// TIA Portal project "PLC_Project" (V17)

(* hardware
DEVICE "S7-1500/ET200MP station_1"  S7-1500 station
   slot 0: "Rail_0"  Rack  6ES7 590-1***0-0AA0
   slot 1: "PLC_1"  CPU 1512C-1 PN  6ES7 512-1CK01-0AB0  V2.9
      slot 3: "CPU display_1"  6ES7591-1AA00-0AA0
      slot 32768: "PROFINET interface_1"  X1
         slot 32769: "Port_1"  X1 P1
         slot 32770: "Port_2"  X1 P2
      slot 34817: "Virtual CP interface port_1"  Virtual CP interface port  Virtual CP interface port
DEVICE "S7-1200 station_1"  S7-1200 Station
   slot 0: "Rack_0"  S7-1200 Rack  Rack  V1.0
   slot 1: "PLC_2"  CPU 1211C DC/DC/DC  6ES7 211-1AD30-0XB0  V2.2
*)

// ===== PLC "PLC_1"  CPU 1512C-1 PN =====

VAR_GLOBAL   // PLC tag table "ControlStep1"
   "highLevelSilo1" AT %Q0.0 : Bool;
   "lowLevelSilo1" AT %Q0.1 : Bool;
   "highLevelSilo2" AT %Q0.2 : Bool;
   "lowLevelSilo2" AT %Q0.3 : Bool;
   "highLevelSilo3" AT %Q0.4 : Bool;
   "lowLevelSilo3" AT %Q0.5 : Bool;
   "highLevelSilo4" AT %Q0.6 : Bool;
   "lowLevelSilo4" AT %Q0.7 : Bool;
   "highLevelSilo5" AT %Q1.0 : Bool;
   "lowLevelSilo5" AT %Q1.1 : Bool;
   "startPumpSilo1" AT %Q1.2 : Bool;
   "stopPumpSilo1" AT %Q1.3 : Bool;
   "startPumpSilo2" AT %Q1.4 : Bool;
   "stopPumpSilo2" AT %Q1.5 : Bool;
   "startPumpSilo3" AT %Q1.6 : Bool;
   "stopPumpSilo3" AT %Q1.7 : Bool;
   "startPumpSilo4" AT %Q2.0 : Bool;
   "stopPumpSilo4" AT %Q2.1 : Bool;
   "startPumpSilo5" AT %Q2.2 : Bool;
   "stopPumpSilo5" AT %Q2.3 : Bool;
   "errorSilo1" AT %I0.0 : Bool;
   "errorSilo2" AT %I0.1 : Bool;
   "errorSilo3" AT %I0.2 : Bool;
   "errorSilo4" AT %I0.3 : Bool;
   "errorSilo5" AT %I0.4 : Bool;
   "levelSilo1" AT %ID5 : Real;
   "levelSilo2" AT %ID10 : Real;
   "levelSilo3" AT %ID14 : Real;
   "levelSilo4" AT %ID18 : Real;
   "levelSilo5" AT %ID22 : Real;
END_VAR

DATA_BLOCK "Recipe"   // DB1
{ S7_Optimized_Access := 'TRUE' }
VERSION : 0.1
   VAR
      maxLevelSilo1 : Real;   // max cua silo 1
      minLevelSilo1 : Real;   // min cua silo 1
      maxLevelSilo2 : Real;   // max cua silo 2
      minLevelSilo2 : Real;   // min cua silo 2
      maxLevelSilo3 : Real;   // max cua silo 3
      minLevelSilo3 : Real;   // min cua silo 3
      maxLevelSilo4 : Real;   // max cua silo 4
      minLevelSilo4 : Real;   // min cua silo 4
      maxLevelSilo5 : Real;   // max cua silo 5
      minLevelSilo5 : Real;   // min cua silo 5
      weightOfRaw1 : Real;   // khoi luong nguyen lieu 1 can thiet
      weightOfRaw2 : Real;   // khoi luong nguyen lieu 2 can thiet
      weightOfRaw3 : Real;   // khoi luong nguyen lieu 3 can thiet
      weightOfSpice : Real;   // khoi luong gia vi can thiet
      weightOfWater : Real;   // khoi luong nuoc can thiet
      errorWeightRaw1 : Real := 2.5;   // sai so khi do khoi luong nguyen lieu 1
      errorWeightRaw2 : Real := 2.5;   // sai so khi do khoi luong nguyen lieu 2
      errorWeightRaw3 : Real := 2.5;   // sai so khi do khoi luong nguyen lieu 3
      errorWeightSpice : Real := 5.0;   // sai so khi do khoi luong gia vi
      errorWeightWater : Real := 7.0;   // sai so khi do khoi luong nuoc
      openValvePercMin : Real := 10.0;   // % mo van nho nhat de ko gap loi co khi
   END_VAR
BEGIN
END_DATA_BLOCK

DATA_BLOCK "Control_DB"   // DB7
{ S7_Optimized_Access := 'TRUE' }
VERSION : 0.1
// stored: InstanceOfName Control
"Control"
BEGIN
END_DATA_BLOCK

DATA_BLOCK "Process_DB"   // DB8
{ S7_Optimized_Access := 'TRUE' }
VERSION : 0.1
// stored: InstanceOfName Process
"Process"
BEGIN
END_DATA_BLOCK

DATA_BLOCK "BtnControl"   // DB10
{ S7_Optimized_Access := 'TRUE' }
VERSION : 0.1
   VAR
      start : Bool;
      stop : Bool;
      auto : Bool;
      manu : Bool;
      reset : Bool;
      pause : Bool;
      resume : Bool;
      restart : Bool;
      hold : Bool;
      emerg : Bool;
      abort : Bool;
      alarm : Bool;
      error : Bool;
      btn_silo1 : Bool;
      btn_silo2 : Bool;
      btn_silo3 : Bool;
      btn_silo4 : Bool;
      btn_silo5 : Bool;
      btn_Conveyor : Bool;
      btn_scaleRaw1 : Bool;
      btn_scaleRaw2 : Bool;
      btn_scaleRaw3 : Bool;
      btn_scaleSpice : Bool;
      btn_scaleWater : Bool;
      btn_runGrinder : Bool;
      btn_runMixer : Bool;
      btn_dischargeSpice : Bool;
      btn_dischargeWater : Bool;
      btn_dischargeMixer : Bool;
      btn_ResetReady : Bool;
   END_VAR
BEGIN
END_DATA_BLOCK

DATA_BLOCK "Data"   // DB11
{ S7_Optimized_Access := 'TRUE' }
VERSION : 0.1
   VAR
      state : Int;
      "step" : Int;
      mode : Int;
      set : Bool;
      targetBatches : Int;
      currentBatches : Int;
      silo1Ready : Bool;
      silo2Ready : Bool;
      silo3Ready : Bool;
      silo4Ready : Bool;
      silo5Ready : Bool;
      spiceReady : Bool;
      waterReady : Bool;
      rawReady : Bool;
      grindDone : Bool;
      mixDone : Bool;
      productReady : Bool;
      resetReadyState : Bool;
      enaPumpSilo1 : Bool;
      enaPumpSilo2 : Bool;
      enaPumpSilo3 : Bool;
      enaPumpSilo4 : Bool;
      enaPumpSilo5 : Bool;
      enaScaleRaw1 : Bool;
      enaScaleRaw2 : Bool;
      enaScaleRaw3 : Bool;
      enaScaleSpice : Bool;
      enaScaleWater : Bool;
      runConveyor : Bool;
      runGrinder : Bool;
      runMixer : Bool;
      enaDischargeSpice : Bool;
      enaDischargeWater : Bool;
      enaDischargeMixer : Bool;
   END_VAR
BEGIN
END_DATA_BLOCK

// folder: DB

DATA_BLOCK "Phase1_DB"   // DB9
{ S7_Optimized_Access := 'TRUE' }
VERSION : 0.1
// stored: InstanceOfName Phase1
"Phase1"
BEGIN
END_DATA_BLOCK

DATA_BLOCK "Phase2_DB"   // DB12
{ S7_Optimized_Access := 'TRUE' }
VERSION : 0.1
// stored: InstanceOfName Phase2
"Phase2"
BEGIN
END_DATA_BLOCK

DATA_BLOCK "Phase3_DB"   // DB13
{ S7_Optimized_Access := 'TRUE' }
VERSION : 0.1
// stored: InstanceOfName Phase3
"Phase3"
BEGIN
END_DATA_BLOCK

DATA_BLOCK "Phase4_DB"   // DB14
{ S7_Optimized_Access := 'TRUE' }
VERSION : 0.1
// stored: InstanceOfName Phase4
"Phase4"
BEGIN
END_DATA_BLOCK

DATA_BLOCK "Phase5_DB"   // DB15
{ S7_Optimized_Access := 'TRUE' }
VERSION : 0.1
// stored: InstanceOfName Phase5
"Phase5"
BEGIN
END_DATA_BLOCK

DATA_BLOCK "Phase6_DB"   // DB16
{ S7_Optimized_Access := 'TRUE' }
VERSION : 0.1
// stored: InstanceOfName Phase6
"Phase6"
BEGIN
END_DATA_BLOCK

DATA_BLOCK "Phase7_DB"   // DB17
{ S7_Optimized_Access := 'TRUE' }
VERSION : 0.1
// stored: InstanceOfName Phase7
"Phase7"
BEGIN
END_DATA_BLOCK

DATA_BLOCK "Phase8_DB"   // DB18
{ S7_Optimized_Access := 'TRUE' }
VERSION : 0.1
// stored: InstanceOfName Phase8
"Phase8"
BEGIN
END_DATA_BLOCK

DATA_BLOCK "Phase9_DB"   // DB19
{ S7_Optimized_Access := 'TRUE' }
VERSION : 0.1
// stored: InstanceOfName Phase9
"Phase9"
BEGIN
END_DATA_BLOCK

DATA_BLOCK "Phase10_DB"   // DB20
{ S7_Optimized_Access := 'TRUE' }
VERSION : 0.1
// stored: InstanceOfName Phase10
"Phase10"
BEGIN
END_DATA_BLOCK

DATA_BLOCK "Phase11_DB"   // DB21
{ S7_Optimized_Access := 'TRUE' }
VERSION : 0.1
// stored: InstanceOfName Phase11
"Phase11"
BEGIN
END_DATA_BLOCK

DATA_BLOCK "Phase12_DB"   // DB22
{ S7_Optimized_Access := 'TRUE' }
VERSION : 0.1
// stored: InstanceOfName Phase12
"Phase12"
BEGIN
END_DATA_BLOCK

DATA_BLOCK "Phase13_DB"   // DB23
{ S7_Optimized_Access := 'TRUE' }
VERSION : 0.1
// stored: InstanceOfName Phase13
"Phase13"
BEGIN
END_DATA_BLOCK

DATA_BLOCK "Phase14_DB"   // DB24
{ S7_Optimized_Access := 'TRUE' }
VERSION : 0.1
// stored: InstanceOfName Phase14
"Phase14"
BEGIN
END_DATA_BLOCK

DATA_BLOCK "Phase15_DB"   // DB25
{ S7_Optimized_Access := 'TRUE' }
VERSION : 0.1
// stored: InstanceOfName Phase15
"Phase15"
BEGIN
END_DATA_BLOCK

DATA_BLOCK "Phase16_DB"   // DB26
{ S7_Optimized_Access := 'TRUE' }
VERSION : 0.1
// stored: InstanceOfName Phase16
"Phase16"
BEGIN
END_DATA_BLOCK

// folder: System blocks/Program resources

DATA_BLOCK "TON_CheckWeight"   // DB2
{ S7_Optimized_Access := 'TRUE' }
AUTHOR : Simatic
FAMILY : IEC
NAME : IEC_TMR
VERSION : 1.0
// stored: InstanceOfName IEC_TIMER
"IEC_TIMER"
BEGIN
END_DATA_BLOCK

DATA_BLOCK "TON_RunGrinder"   // DB3
{ S7_Optimized_Access := 'TRUE' }
AUTHOR : Simatic
FAMILY : IEC
NAME : IEC_TMR
VERSION : 1.0
// stored: InstanceOfName IEC_TIMER
"IEC_TIMER"
BEGIN
END_DATA_BLOCK

DATA_BLOCK "TON_RunMixer"   // DB4
{ S7_Optimized_Access := 'TRUE' }
AUTHOR : Simatic
FAMILY : IEC
NAME : IEC_TMR
VERSION : 1.0
// stored: InstanceOfName IEC_TIMER
"IEC_TIMER"
BEGIN
END_DATA_BLOCK

DATA_BLOCK "TON_ResetReadyState"   // DB5
{ S7_Optimized_Access := 'TRUE' }
AUTHOR : Simatic
FAMILY : IEC
NAME : IEC_TMR
VERSION : 1.0
// stored: InstanceOfName IEC_TIMER
"IEC_TIMER"
BEGIN
END_DATA_BLOCK

DATA_BLOCK "TP_ResetReadyState"   // DB6
{ S7_Optimized_Access := 'TRUE' }
AUTHOR : Simatic
FAMILY : IEC
NAME : IEC_TMR
VERSION : 1.0
// stored: InstanceOfName IEC_TIMER
"IEC_TIMER"
BEGIN
END_DATA_BLOCK

DATA_BLOCK "TOn_CheckWeightRaw3"   // DB27
{ S7_Optimized_Access := 'TRUE' }
AUTHOR : Simatic
FAMILY : IEC
NAME : IEC_TMR
VERSION : 1.0
// stored: InstanceOfName IEC_TIMER
"IEC_TIMER"
BEGIN
END_DATA_BLOCK

DATA_BLOCK "IEC_Timer_0_DB"   // DB28
{ S7_Optimized_Access := 'TRUE' }
AUTHOR : Simatic
FAMILY : IEC
NAME : IEC_TMR
VERSION : 1.0
// stored: InstanceOfName IEC_TIMER
"IEC_TIMER"
BEGIN
END_DATA_BLOCK

// folder: (top level)

FUNCTION_BLOCK "Control"   // FB1, SCL
{ S7_Optimized_Access := 'TRUE' }
VERSION : 0.1
   VAR_INPUT
      start : Bool;
      stop : Bool;
      auto : Bool;
      manu : Bool;
      reset : Bool;
      pause : Bool;
      resume : Bool;
      restart : Bool;
      hold : Bool;
      emerg : Bool;
      abort : Bool;
      alarm : Bool;
      error : Bool;
   END_VAR
   VAR_IN_OUT
      mode : Int;
      state : Int;
      "step" : Int;
   END_VAR
BEGIN
   //chon che do hoat dong
   IF #state = 0 THEN
       IF (#auto AND #manu) OR (NOT #auto AND NOT #manu) THEN
           #mode := 0;
       ELSE
           IF #auto THEN
               #mode := 1;
           END_IF;
           IF #manu THEN
               #mode := 2;
           END_IF;
       END_IF;
   END_IF;

   IF #mode <> 0 THEN
       CASE #state OF
           0:
               IF #start THEN
                   #state := 1;
               END_IF;
           1:
               IF #abort THEN
                   #state := 2;
               ELSIF #stop THEN
                   #state := 3;
               ELSIF #pause THEN
                   #state := 4;
               ELSIF #hold THEN
                   #state := 5;
               ELSIF #step = 6 THEN
                   #state := 6;
               END_IF;
           2, 3, 6:
               IF #reset THEN
                   #state := 0;
               END_IF;
           4:
               IF #resume THEN
                   #state := 1;
               END_IF;
           5:
               IF #restart THEN
                   #state := 1;
               END_IF;

       END_CASE;
   END_IF;
END_FUNCTION_BLOCK

FUNCTION_BLOCK "Process"   // FB2, SCL
{ S7_Optimized_Access := 'TRUE' }
VERSION : 0.1
   VAR_INPUT
      state : Int;   // trang thai hoat dong
      mode : Int;   // che do hoat dong, 1: auto, 2: manu
      set : Bool;   // tin hieu set cac thong so cai dat
      targetBatches : Int;   // So luong me can lam
      currentBatches : Int;   // So luong me hien tai
      silo1Ready : Bool;   // silo 1 da san sang cung cap nguyen lieu
      silo2Ready : Bool;   // silo 2 da san sang cung cap nguyen lieu
      silo3Ready : Bool;   // silo 3 da san sang cung cap nguyen lieu
      silo4Ready : Bool;   // silo 4 da san sang cung cap gia vi
      silo5Ready : Bool;   // silo 5 da san sang cung cap nuoc
      spiceReady : Bool;   // da can xong gia vi
      waterReady : Bool;   // da can xong nuoc
      rawReady : Bool;   // da can xong va dua nguyen lieu vao bon nghien
      grindDone : Bool;   // da nghien xong nguyen lieu
      mixDone : Bool;   // da tron xong nguyen lieu
      productReady : Bool;
      btn_resetReady : Bool;   // dkhien reset trang thai ready bang tay (mode manu)
      btn_silo1 : Bool;   // dkhien silo bang tay (mode manu)
      btn_silo2 : Bool;   // dkhien silo bang tay (mode manu)
      btn_silo3 : Bool;   // dkhien silo bang tay (mode manu)
      btn_silo4 : Bool;   // dkhien silo bang tay (mode manu)
      btn_silo5 : Bool;   // dkhien silo bang tay (mode manu)
      btn_runConveyor : Bool;   // dkhien can nguyen lieu bang tay (mode manu)
      btn_scaleRaw1 : Bool;   // xa nguyen lieu raw 1 xuong bang tai bang tay (mode manu)
      btn_scaleRaw2 : Bool;   // xa nguyen lieu raw 2 xuong bang tai bang tay (mode manu)
      btn_scaleRaw3 : Bool;   // xa nguyen lieu raw 3 xuong bang tai bang tay (mode manu)
      btn_scaleSpice : Bool;   // dkhien can gia vi bang tay (mode manu)
      btn_scaleWater : Bool;   // dkhien can nuoc bang tay (mode manu)
      btn_runGrinder : Bool;   // dkhien chay may nghien bang tay (mode manu)
      btn_runMixer : Bool;   // dkhien chay may tron bang tay (mode manu)
      btn_DischargeSpice : Bool;   // dkhien van gia vi bang tay (mode manu)
      btn_DischargeWater : Bool;   // dkhien van nuoc bang tay (mode manu)
      btn_DischargeMixer : Bool;   // dkhien van tron bang tay (mode manu)
   END_VAR
   VAR_OUTPUT
      resetReadyState : Bool;   // tiep tuc lam me moi -> reset lai cac bien ready
      enaPumpSilo1 : Bool;   // cho phep bon 1 bat dau hoat dong
      enaPumpSilo2 : Bool;   // cho phep bon 2 bat dau hoat dong
      enaPumpSilo3 : Bool;   // cho phep bon 3 bat dau hoat dong
      enaPumpSilo4 : Bool;   // cho phep bon 4 bat dau hoat dong
      enaPumpSilo5 : Bool;   // cho phep bon 5 bat dau hoat dong
      enaScaleRaw1 : Bool;
      enaScaleRaw2 : Bool;
      enaScaleRaw3 : Bool;
      enaScaleSpice : Bool;   // cho phep can gia vi
      enaScaleWater : Bool;   // cho phep can nuoc
      runConveyor : Bool;   // chay bang tai
      runGrinder : Bool;   // chay may nghien
      runMixer : Bool;   // chay may tron
      enaDischargeSpice : Bool;   // cho phep xa van gia vi vao may tron
      enaDischargeWater : Bool;   // cho phep xa van nuoc vao may tron
      enaDischargeMixer : Bool;   // cho phep xa hon ho[p da tron -> hoan thanh 1 batch
   END_VAR
   VAR_IN_OUT
      "step" : Int;
   END_VAR
BEGIN
   IF #state = 1 AND #mode = 1 AND #set THEN
       IF #step = 0 AND #currentBatches < #targetBatches THEN
           #step := 1;
       END_IF;

       CASE #step OF
           1: 
               #enaPumpSilo1 := TRUE;
               #enaPumpSilo2 := TRUE;
               #enaPumpSilo3 := TRUE;
               #enaPumpSilo4 := TRUE;
               #enaPumpSilo5 := TRUE;
               IF #silo1Ready AND #silo2Ready AND #silo3Ready AND #silo4Ready AND #silo5Ready THEN
                   #enaPumpSilo1 := FALSE;
                   #enaPumpSilo2 := FALSE;
                   #enaPumpSilo3 := FALSE;
                   #enaPumpSilo4 := FALSE;
                   #enaPumpSilo5 := FALSE;
                   #step := 2;
               END_IF;

           2: 
               #runConveyor := TRUE;
               #enaScaleRaw1 := TRUE;
               #enaScaleRaw2 := TRUE;
               #enaScaleRaw3 := TRUE;
               #enaScaleWater := TRUE;
               #enaScaleSpice := TRUE;
               IF #rawReady AND #spiceReady AND #waterReady THEN
                   #runConveyor := FALSE;
                   #enaScaleRaw1 := FALSE;
                   #enaScaleRaw2 := FALSE;
                   #enaScaleRaw3 := FALSE;
                   #enaScaleWater := FALSE;
                   #enaScaleSpice := FALSE;
                   #step := 3;
               END_IF;

           3:
               #runGrinder := TRUE;
               IF #grindDone THEN
                   #runGrinder := FALSE;
                   #step := 4;
               END_IF;

           4: 
               #runMixer := TRUE;
               #enaDischargeWater := TRUE; //cho phep mo van, mo bao nhieu % tuy thuoc vao phase 14, 15 quyet dinh
               #enaDischargeSpice := TRUE;
               IF #mixDone THEN
                   #runMixer := FALSE;
                   #enaDischargeWater := FALSE;
                   #enaDischargeSpice := FALSE;
                   #step := 5;
               END_IF;

           5: 
               #enaDischargeMixer := TRUE;
               IF NOT #productReady THEN
                   #currentBatches := #currentBatches + 1;
                   #enaDischargeMixer := FALSE;
                   #step := 0;
               END_IF;
               // reset cac bien ready ve FALSE trong 1s -> chac chan bien nao cung dc reset
               "TP_ResetReadyState".TP(IN := NOT #productReady,
                                       PT := T#1000ms,
                                       Q => #resetReadyState);
       END_CASE;

   ELSIF #state = 1 AND #mode = 2 AND #set THEN
       #step := 0;
       #resetReadyState := #btn_resetReady;
           //Dk silo
           #enaPumpSilo1 := #btn_silo1;
           #enaPumpSilo2 := #btn_silo2;
           #enaPumpSilo3 := #btn_silo3;
           #enaPumpSilo4 := #btn_silo4;
           #enaPumpSilo5 := #btn_silo5;

           //Dk can va bang tai 
           #runConveyor := #btn_runConveyor;
           #enaScaleRaw1 := #btn_scaleRaw1;
           #enaScaleRaw2 := #btn_scaleRaw2;
           #enaScaleRaw3 := #btn_scaleRaw3;
           #enaScaleWater := #btn_scaleWater;
           #enaScaleSpice := #btn_scaleWater;

           //Dk may nghien va may tron
           #runGrinder := #btn_runGrinder;
           #runMixer := #btn_runMixer;

           //Dong/mo van
           #enaDischargeWater := #btn_DischargeWater;
           #enaDischargeSpice := #btn_DischargeSpice;
           #enaDischargeMixer := #btn_DischargeMixer;
   END_IF;
END_FUNCTION_BLOCK

ORGANIZATION_BLOCK "Main"   // OB1, LAD, ProgramCycle
TITLE = "Main Program Sweep (Cycle)"
{ S7_Optimized_Access := 'TRUE' }
VERSION : 0.1
   VAR_INPUT
      Initial_Call : Bool;   // Initial call of this OB
      Remanence : Bool;   // =True, if remanent data are available
   END_VAR
   VAR_TEMP   // added for the SCL form of the ladder/FBD networks
      _w1 : Bool;
      _w2 : Bool;
   END_VAR
BEGIN

REGION Network 1
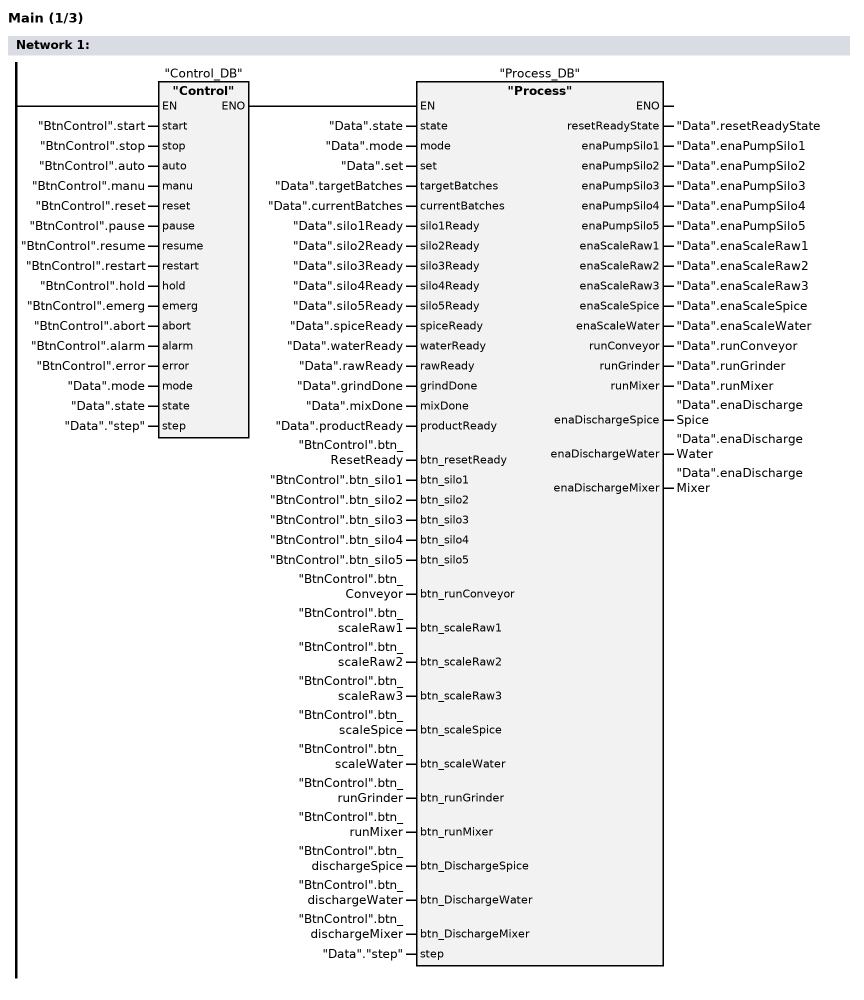
   RUNG wire#powerrail
      "Control_DB"(start := "BtnControl".start, stop := "BtnControl".stop, auto := "BtnControl".auto, manu := "BtnControl".manu, reset := "BtnControl".reset, pause := "BtnControl".pause, resume := "BtnControl".resume, restart := "BtnControl".restart, hold := "BtnControl".hold, emerg := "BtnControl".emerg, abort := "BtnControl".abort, alarm := "BtnControl".alarm, error := "BtnControl".error, mode := "Data".mode, state := "Data".state, "step" := "Data"."step")
      "Process_DB"(state := "Data".state, mode := "Data".mode, set := "Data".set, targetBatches := "Data".targetBatches, currentBatches := "Data".currentBatches, silo1Ready := "Data".silo1Ready, silo2Ready := "Data".silo2Ready, silo3Ready := "Data".silo3Ready, silo4Ready := "Data".silo4Ready, silo5Ready := "Data".silo5Ready, spiceReady := "Data".spiceReady, waterReady := "Data".waterReady, rawReady := "Data".rawReady, grindDone := "Data".grindDone, mixDone := "Data".mixDone, productReady := "Data".productReady, btn_resetReady := "BtnControl".btn_ResetReady, btn_silo1 := "BtnControl".btn_silo1, btn_silo2 := "BtnControl".btn_silo2, btn_silo3 := "BtnControl".btn_silo3, btn_silo4 := "BtnControl".btn_silo4, btn_silo5 := "BtnControl".btn_silo5, btn_runConveyor := "BtnControl".btn_Conveyor, btn_scaleRaw1 := "BtnControl".btn_scaleRaw1, btn_scaleRaw2 := "BtnControl".btn_scaleRaw2, btn_scaleRaw3 := "BtnControl".btn_scaleRaw3, btn_scaleSpice := "BtnControl".btn_scaleSpice, btn_scaleWater := "BtnControl".btn_scaleWater, btn_runGrinder := "BtnControl".btn_runGrinder, btn_runMixer := "BtnControl".btn_runMixer, btn_DischargeSpice := "BtnControl".btn_dischargeSpice, btn_DischargeWater := "BtnControl".btn_dischargeWater, btn_DischargeMixer := "BtnControl".btn_dischargeMixer, "step" := "Data"."step", resetReadyState => "Data".resetReadyState, enaPumpSilo1 => "Data".enaPumpSilo1, enaPumpSilo2 => "Data".enaPumpSilo2, enaPumpSilo3 => "Data".enaPumpSilo3, enaPumpSilo4 => "Data".enaPumpSilo4, enaPumpSilo5 => "Data".enaPumpSilo5, enaScaleRaw1 => "Data".enaScaleRaw1, enaScaleRaw2 => "Data".enaScaleRaw2, enaScaleRaw3 => "Data".enaScaleRaw3, enaScaleSpice => "Data".enaScaleSpice, enaScaleWater => "Data".enaScaleWater, runConveyor => "Data".runConveyor, runGrinder => "Data".runGrinder, runMixer => "Data".runMixer, enaDischargeSpice => "Data".enaDischargeSpice, enaDischargeWater => "Data".enaDischargeWater, enaDischargeMixer => "Data".enaDischargeMixer)
   END_RUNG
   // the same network as SCL:
   "Control_DB"(start := "BtnControl".start,   // "Control"
                stop := "BtnControl".stop,
                auto := "BtnControl".auto,
                manu := "BtnControl".manu,
                reset := "BtnControl".reset,
                pause := "BtnControl".pause,
                resume := "BtnControl".resume,
                restart := "BtnControl".restart,
                hold := "BtnControl".hold,
                emerg := "BtnControl".emerg,
                abort := "BtnControl".abort,
                alarm := "BtnControl".alarm,
                error := "BtnControl".error,
                mode := "Data".mode,
                state := "Data".state,
                "step" := "Data"."step",
                ENO => #_w1);
   IF #_w1 THEN
       "Process_DB"(state := "Data".state,   // "Process"
                    mode := "Data".mode,
                    set := "Data".set,
                    targetBatches := "Data".targetBatches,
                    currentBatches := "Data".currentBatches,
                    silo1Ready := "Data".silo1Ready,
                    silo2Ready := "Data".silo2Ready,
                    silo3Ready := "Data".silo3Ready,
                    silo4Ready := "Data".silo4Ready,
                    silo5Ready := "Data".silo5Ready,
                    spiceReady := "Data".spiceReady,
                    waterReady := "Data".waterReady,
                    rawReady := "Data".rawReady,
                    grindDone := "Data".grindDone,
                    mixDone := "Data".mixDone,
                    productReady := "Data".productReady,
                    btn_resetReady := "BtnControl".btn_ResetReady,
                    btn_silo1 := "BtnControl".btn_silo1,
                    btn_silo2 := "BtnControl".btn_silo2,
                    btn_silo3 := "BtnControl".btn_silo3,
                    btn_silo4 := "BtnControl".btn_silo4,
                    btn_silo5 := "BtnControl".btn_silo5,
                    btn_runConveyor := "BtnControl".btn_Conveyor,
                    btn_scaleRaw1 := "BtnControl".btn_scaleRaw1,
                    btn_scaleRaw2 := "BtnControl".btn_scaleRaw2,
                    btn_scaleRaw3 := "BtnControl".btn_scaleRaw3,
                    btn_scaleSpice := "BtnControl".btn_scaleSpice,
                    btn_scaleWater := "BtnControl".btn_scaleWater,
                    btn_runGrinder := "BtnControl".btn_runGrinder,
                    btn_runMixer := "BtnControl".btn_runMixer,
                    btn_DischargeSpice := "BtnControl".btn_dischargeSpice,
                    btn_DischargeWater := "BtnControl".btn_dischargeWater,
                    btn_DischargeMixer := "BtnControl".btn_dischargeMixer,
                    "step" := "Data"."step",
                    resetReadyState => "Data".resetReadyState,
                    enaPumpSilo1 => "Data".enaPumpSilo1,
                    enaPumpSilo2 => "Data".enaPumpSilo2,
                    enaPumpSilo3 => "Data".enaPumpSilo3,
                    enaPumpSilo4 => "Data".enaPumpSilo4,
                    enaPumpSilo5 => "Data".enaPumpSilo5,
                    enaScaleRaw1 => "Data".enaScaleRaw1,
                    enaScaleRaw2 => "Data".enaScaleRaw2,
                    enaScaleRaw3 => "Data".enaScaleRaw3,
                    enaScaleSpice => "Data".enaScaleSpice,
                    enaScaleWater => "Data".enaScaleWater,
                    runConveyor => "Data".runConveyor,
                    runGrinder => "Data".runGrinder,
                    runMixer => "Data".runMixer,
                    enaDischargeSpice => "Data".enaDischargeSpice,
                    enaDischargeWater => "Data".enaDischargeWater,
                    enaDischargeMixer => "Data".enaDischargeMixer);
   END_IF;
END_REGION

REGION Network 2
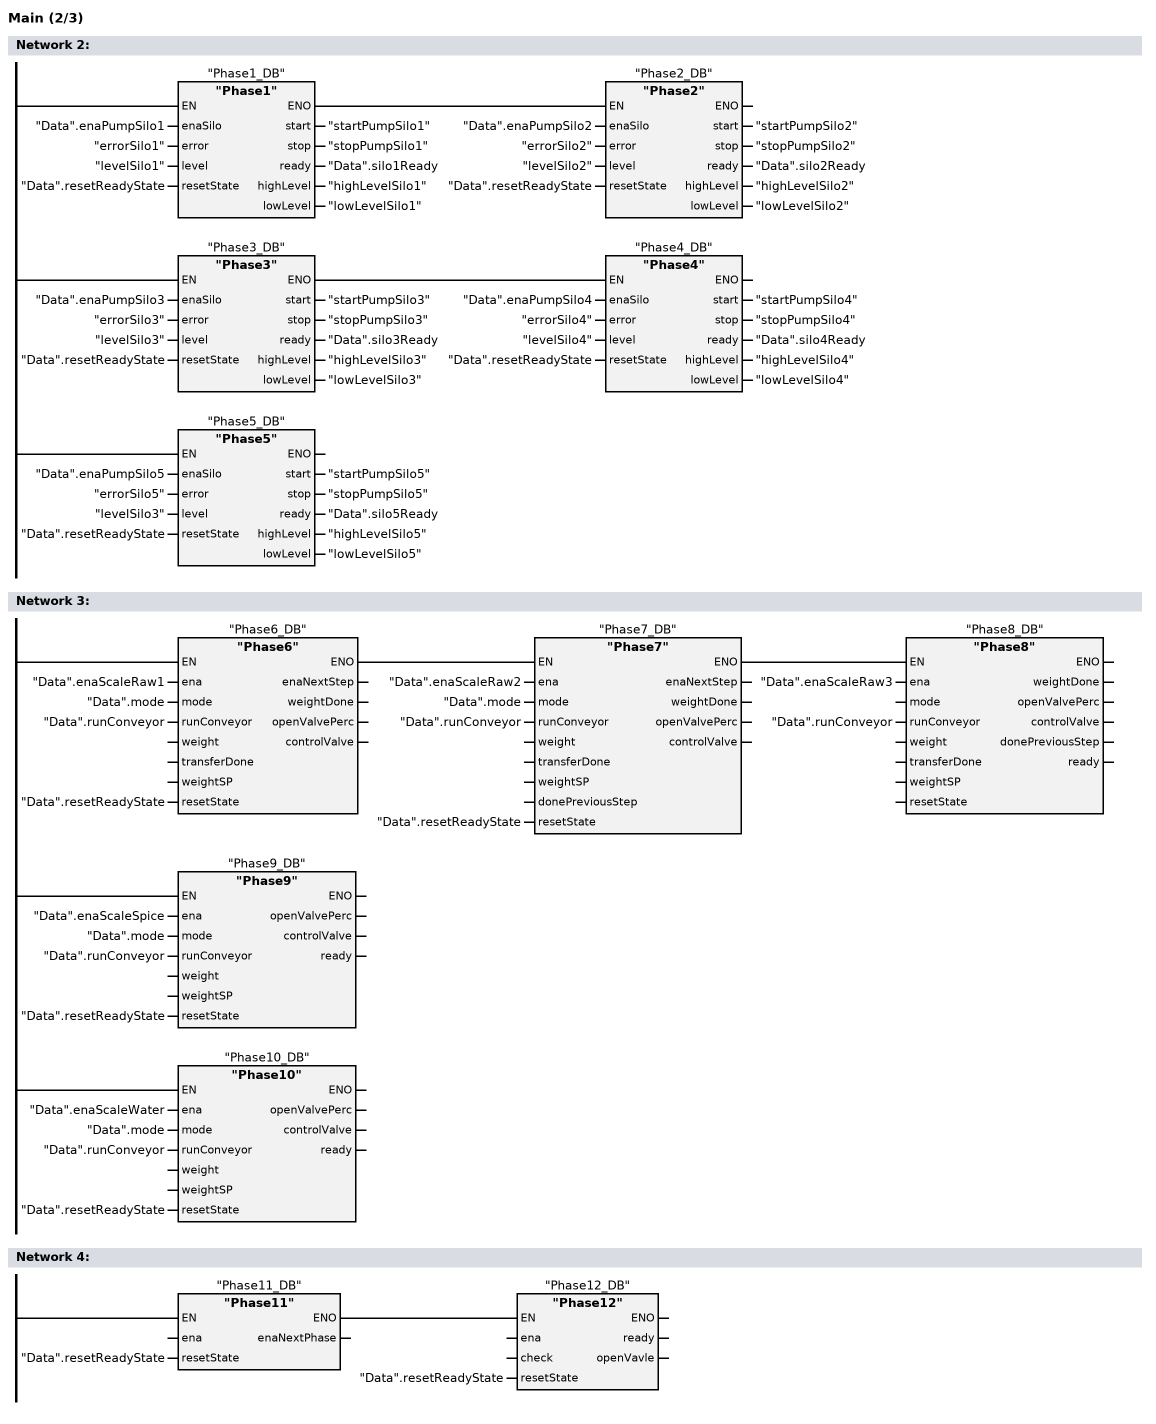
   RUNG wire#powerrail
      "Phase1_DB"(enaSilo := "Data".enaPumpSilo1, error := "errorSilo1", level := "levelSilo1", resetState := "Data".resetReadyState, start => "startPumpSilo1", stop => "stopPumpSilo1", ready => "Data".silo1Ready, highLevel => "highLevelSilo1", lowLevel => "lowLevelSilo1")
      "Phase2_DB"(enaSilo := "Data".enaPumpSilo2, error := "errorSilo2", level := "levelSilo2", resetState := "Data".resetReadyState, start => "startPumpSilo2", stop => "stopPumpSilo2", ready => "Data".silo2Ready, highLevel => "highLevelSilo2", lowLevel => "lowLevelSilo2")
   END_RUNG
   RUNG wire#powerrail
      "Phase3_DB"(enaSilo := "Data".enaPumpSilo3, error := "errorSilo3", level := "levelSilo3", resetState := "Data".resetReadyState, start => "startPumpSilo3", stop => "stopPumpSilo3", ready => "Data".silo3Ready, highLevel => "highLevelSilo3", lowLevel => "lowLevelSilo3")
      "Phase4_DB"(enaSilo := "Data".enaPumpSilo4, error := "errorSilo4", level := "levelSilo4", resetState := "Data".resetReadyState, start => "startPumpSilo4", stop => "stopPumpSilo4", ready => "Data".silo4Ready, highLevel => "highLevelSilo4", lowLevel => "lowLevelSilo4")
   END_RUNG
   RUNG wire#powerrail
      "Phase5_DB"(enaSilo := "Data".enaPumpSilo5, error := "errorSilo5", level := "levelSilo3", resetState := "Data".resetReadyState, start => "startPumpSilo5", stop => "stopPumpSilo5", ready => "Data".silo5Ready, highLevel => "highLevelSilo5", lowLevel => "lowLevelSilo5")
   END_RUNG
   // the same network as SCL:
   "Phase1_DB"(enaSilo := "Data".enaPumpSilo1,   // "Phase1"
               error := "errorSilo1",
               level := "levelSilo1",
               resetState := "Data".resetReadyState,
               start => "startPumpSilo1",
               stop => "stopPumpSilo1",
               ready => "Data".silo1Ready,
               highLevel => "highLevelSilo1",
               lowLevel => "lowLevelSilo1",
               ENO => #_w1);
   IF #_w1 THEN
       "Phase2_DB"(enaSilo := "Data".enaPumpSilo2,   // "Phase2"
                   error := "errorSilo2",
                   level := "levelSilo2",
                   resetState := "Data".resetReadyState,
                   start => "startPumpSilo2",
                   stop => "stopPumpSilo2",
                   ready => "Data".silo2Ready,
                   highLevel => "highLevelSilo2",
                   lowLevel => "lowLevelSilo2");
   END_IF;
   "Phase3_DB"(enaSilo := "Data".enaPumpSilo3,   // "Phase3"
               error := "errorSilo3",
               level := "levelSilo3",
               resetState := "Data".resetReadyState,
               start => "startPumpSilo3",
               stop => "stopPumpSilo3",
               ready => "Data".silo3Ready,
               highLevel => "highLevelSilo3",
               lowLevel => "lowLevelSilo3",
               ENO => #_w2);
   IF #_w2 THEN
       "Phase4_DB"(enaSilo := "Data".enaPumpSilo4,   // "Phase4"
                   error := "errorSilo4",
                   level := "levelSilo4",
                   resetState := "Data".resetReadyState,
                   start => "startPumpSilo4",
                   stop => "stopPumpSilo4",
                   ready => "Data".silo4Ready,
                   highLevel => "highLevelSilo4",
                   lowLevel => "lowLevelSilo4");
   END_IF;
   "Phase5_DB"(enaSilo := "Data".enaPumpSilo5,   // "Phase5"
               error := "errorSilo5",
               level := "levelSilo3",
               resetState := "Data".resetReadyState,
               start => "startPumpSilo5",
               stop => "stopPumpSilo5",
               ready => "Data".silo5Ready,
               highLevel => "highLevelSilo5",
               lowLevel => "lowLevelSilo5");
END_REGION

REGION Network 3
   RUNG wire#powerrail
      "Phase6_DB"(ena := "Data".enaScaleRaw1, mode := "Data".mode, runConveyor := "Data".runConveyor, weight :=, transferDone :=, weightSP :=, resetState := "Data".resetReadyState, enaNextStep =>, weightDone =>, openValvePerc =>, controlValve =>)
      "Phase7_DB"(ena := "Data".enaScaleRaw2, mode := "Data".mode, runConveyor := "Data".runConveyor, weight :=, transferDone :=, weightSP :=, donePreviousStep :=, resetState := "Data".resetReadyState, enaNextStep =>, weightDone =>, openValvePerc =>, controlValve =>)
      "Phase8_DB"(ena := "Data".enaScaleRaw3, mode :=, runConveyor := "Data".runConveyor, weight :=, transferDone :=, weightSP :=, resetState :=, weightDone =>, openValvePerc =>, controlValve =>, donePreviousStep =>, ready =>)
   END_RUNG
   RUNG wire#powerrail
      "Phase9_DB"(ena := "Data".enaScaleSpice, mode := "Data".mode, runConveyor := "Data".runConveyor, weight :=, weightSP :=, resetState := "Data".resetReadyState, openValvePerc =>, controlValve =>, ready =>)
   END_RUNG
   RUNG wire#powerrail
      "Phase10_DB"(ena := "Data".enaScaleWater, mode := "Data".mode, runConveyor := "Data".runConveyor, weight :=, weightSP :=, resetState := "Data".resetReadyState, openValvePerc =>, controlValve =>, ready =>)
   END_RUNG
   // the same network as SCL:
   "Phase6_DB"(ena := "Data".enaScaleRaw1,   // "Phase6"
               mode := "Data".mode,
               runConveyor := "Data".runConveyor,
               resetState := "Data".resetReadyState,
               ENO => #_w1);
   "Phase7_DB"(EN := #_w1,   // "Phase7"
               ena := "Data".enaScaleRaw2,
               mode := "Data".mode,
               runConveyor := "Data".runConveyor,
               resetState := "Data".resetReadyState,
               ENO => #_w2);
   IF #_w2 THEN
       "Phase8_DB"(ena := "Data".enaScaleRaw3, runConveyor := "Data".runConveyor);   // "Phase8"
   END_IF;
   "Phase9_DB"(ena := "Data".enaScaleSpice,   // "Phase9"
               mode := "Data".mode,
               runConveyor := "Data".runConveyor,
               resetState := "Data".resetReadyState);
   "Phase10_DB"(ena := "Data".enaScaleWater,   // "Phase10"
                mode := "Data".mode,
                runConveyor := "Data".runConveyor,
                resetState := "Data".resetReadyState);
END_REGION

REGION Network 4
   RUNG wire#powerrail
      "Phase11_DB"(ena :=, resetState := "Data".resetReadyState, enaNextPhase =>)
      "Phase12_DB"(ena :=, check :=, resetState := "Data".resetReadyState, ready =>, openVavle =>)
   END_RUNG
   // the same network as SCL:
   "Phase11_DB"(resetState := "Data".resetReadyState, ENO => #_w1);   // "Phase11"
   IF #_w1 THEN
       "Phase12_DB"(resetState := "Data".resetReadyState);   // "Phase12"
   END_IF;
END_REGION

REGION Network 5
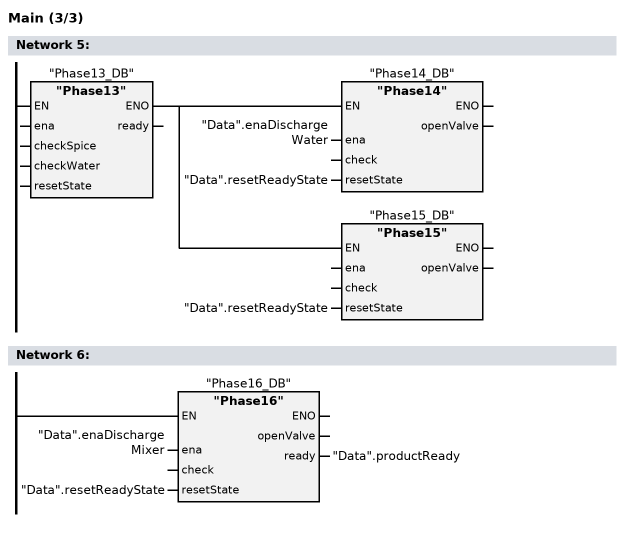
   RUNG wire#powerrail
      "Phase13_DB"(ena :=, checkSpice :=, checkWater :=, resetState :=, ready =>)
      wire#w1
      "Phase14_DB"(ena := "Data".enaDischargeWater, check :=, resetState := "Data".resetReadyState, openValve =>)
   END_RUNG
   RUNG wire#w1
      "Phase15_DB"(ena :=, check :=, resetState := "Data".resetReadyState, openValve =>)
   END_RUNG
   // the same network as SCL:
   "Phase13_DB"(ENO => #_w1);   // "Phase13"
   IF #_w1 THEN
       "Phase14_DB"(ena := "Data".enaDischargeWater, resetState := "Data".resetReadyState);   // "Phase14"
       "Phase15_DB"(resetState := "Data".resetReadyState);   // "Phase15"
   END_IF;
END_REGION

REGION Network 6
   RUNG wire#powerrail
      "Phase16_DB"(ena := "Data".enaDischargeMixer, check :=, resetState := "Data".resetReadyState, openValve =>, ready => "Data".productReady)
   END_RUNG
   // the same network as SCL:
   "Phase16_DB"(ena := "Data".enaDischargeMixer,   // "Phase16"
                resetState := "Data".resetReadyState,
                ready => "Data".productReady);
END_REGION
END_ORGANIZATION_BLOCK

// folder: Unit1(prepareSilo1_Raw)

FUNCTION_BLOCK "Phase1"   // FB3, SCL
{ S7_Optimized_Access := 'TRUE' }
VERSION : 0.1
   VAR_INPUT
      enaSilo : Bool;
      error : Bool;
      level : Real;
      resetState : Bool;
   END_VAR
   VAR_OUTPUT
      start : Bool;
      stop : Bool;
      ready : Bool;
      highLevel : Bool;
      lowLevel : Bool;
   END_VAR
BEGIN
   #highLevel := #level >= "Recipe".maxLevelSilo1;
   #lowLevel := #level <= "Recipe".minLevelSilo1;
   #start := #enaSilo AND #lowLevel;
   #stop := #highLevel OR #error;
   #ready := NOT #highLevel AND NOT #lowLevel;
   IF #resetState THEN
       #ready := FALSE;
   END_IF;
END_FUNCTION_BLOCK

// folder: Unit10(mixAndDone)

FUNCTION_BLOCK "Phase13"   // FB15, SCL
{ S7_Optimized_Access := 'TRUE' }
VERSION : 0.1
   VAR_INPUT
      ena : Bool;   // cho phep hoat dong mixer
      checkSpice : Bool;   // ktra da co du gia vi trong bon chua
      checkWater : Bool;   // ktra da co du nuoc trong bon chua
      resetState : Bool;
   END_VAR
   VAR_OUTPUT
      ready : Bool;
   END_VAR
   VAR CONSTANT
      "time" : Time := T#10s;
   END_VAR
BEGIN
       "TON_RunMixer".TON(IN := #ena AND #checkSpice AND #checkWater,
                          PT := #time,
                          Q => #ready);
       IF #resetState THEN
           #ready := FALSE;
       END_IF;
END_FUNCTION_BLOCK

FUNCTION_BLOCK "Phase14"   // FB16, SCL
{ S7_Optimized_Access := 'TRUE' }
VERSION : 0.1
   VAR_INPUT
      ena : Bool;
      check : Bool;   // ktra bon con gia vi ko
      resetState : Bool;
   END_VAR
   VAR_OUTPUT
      openValve : Bool;
   END_VAR
BEGIN
   IF #ena THEN
       #openValve := TRUE;
       IF NOT #check THEN
           #openValve := FALSE;
       END_IF;
   END_IF;
END_FUNCTION_BLOCK

FUNCTION_BLOCK "Phase15"   // FB17, SCL
{ S7_Optimized_Access := 'TRUE' }
VERSION : 0.1
   VAR_INPUT
      ena : Bool;
      check : Bool;   // ktra bon con nuoc ko
      resetState : Bool;
   END_VAR
   VAR_OUTPUT
      openValve : Bool;
   END_VAR
BEGIN
   IF #ena THEN
       #openValve := TRUE;
       IF NOT #check THEN
           #openValve := FALSE;
       END_IF;
   END_IF;
END_FUNCTION_BLOCK

FUNCTION_BLOCK "Phase16"   // FB18, SCL
{ S7_Optimized_Access := 'TRUE' }
VERSION : 0.1
   VAR_INPUT
      ena : Bool;
      check : Bool;   // ktra hon hop con trong bon ko
      resetState : Bool;
   END_VAR
   VAR_OUTPUT
      openValve : Bool;
      ready : Bool;
   END_VAR
BEGIN
   IF #ena THEN
       #openValve := TRUE;
       IF NOT #check THEN
           #openValve := FALSE;
           #ready := TRUE;
       END_IF;
   END_IF;

   IF #resetState THEN
       #ready := FALSE;
   END_IF;
END_FUNCTION_BLOCK

// folder: Unit2(prepareSilo2_Raw)

FUNCTION_BLOCK "Phase2"   // FB4, SCL
{ S7_Optimized_Access := 'TRUE' }
VERSION : 0.1
   VAR_INPUT
      enaSilo : Bool;
      error : Bool;
      level : Real;
      resetState : Bool;
   END_VAR
   VAR_OUTPUT
      start : Bool;
      stop : Bool;
      ready : Bool;
      highLevel : Bool;
      lowLevel : Bool;
   END_VAR
BEGIN
   #highLevel := #level >= "Recipe".maxLevelSilo2;
   #lowLevel := #level <= "Recipe".minLevelSilo2;
   #start := #enaSilo AND #lowLevel;
   #stop := #highLevel OR #error;
   #ready := NOT #highLevel AND NOT #lowLevel;
   IF #resetState THEN
       #ready := FALSE;
   END_IF;
END_FUNCTION_BLOCK

// folder: Unit3(prepareSilo3_Raw)

FUNCTION_BLOCK "Phase3"   // FB5, SCL
{ S7_Optimized_Access := 'TRUE' }
VERSION : 0.1
   VAR_INPUT
      enaSilo : Bool;
      error : Bool;
      level : Real;
      resetState : Bool;
   END_VAR
   VAR_OUTPUT
      start : Bool;
      stop : Bool;
      ready : Bool;
      highLevel : Bool;
      lowLevel : Bool;
   END_VAR
BEGIN
   #highLevel := #level >= "Recipe".maxLevelSilo3;
   #lowLevel := #level <= "Recipe".minLevelSilo3;
   #start := #enaSilo AND #lowLevel;
   #stop := #highLevel OR #error;
   #ready := NOT #highLevel AND NOT #lowLevel;
   IF #resetState THEN
       #ready := FALSE;
   END_IF;
END_FUNCTION_BLOCK

// folder: Unit4(prepareSilo4_Spice)

FUNCTION_BLOCK "Phase4"   // FB6, SCL
{ S7_Optimized_Access := 'TRUE' }
VERSION : 0.1
   VAR_INPUT
      enaSilo : Bool;
      error : Bool;
      level : Real;
      resetState : Bool;
   END_VAR
   VAR_OUTPUT
      start : Bool;
      stop : Bool;
      ready : Bool;
      highLevel : Bool;
      lowLevel : Bool;
   END_VAR
BEGIN
   #highLevel := #level >= "Recipe".maxLevelSilo4;
   #lowLevel := #level <= "Recipe".minLevelSilo4;
   #start := #enaSilo AND #lowLevel;
   #stop := #highLevel OR #error;
   #ready := NOT #highLevel AND NOT #lowLevel;
   IF #resetState THEN
       #ready := FALSE;
   END_IF;
END_FUNCTION_BLOCK

// folder: Unit5(prepareSilo5_Water)

FUNCTION_BLOCK "Phase5"   // FB7, SCL
{ S7_Optimized_Access := 'TRUE' }
VERSION : 0.1
   VAR_INPUT
      enaSilo : Bool;
      error : Bool;
      level : Real;
      resetState : Bool;
   END_VAR
   VAR_OUTPUT
      start : Bool;
      stop : Bool;
      ready : Bool;
      highLevel : Bool;
      lowLevel : Bool;
   END_VAR
BEGIN
   #highLevel := #level >= "Recipe".maxLevelSilo5;
   #lowLevel := #level <= "Recipe".minLevelSilo5;
   #start := #enaSilo AND #lowLevel;
   #stop := #highLevel OR #error;
   #ready := NOT #highLevel AND NOT #lowLevel;
   IF #resetState THEN
       #ready := FALSE;
   END_IF;
END_FUNCTION_BLOCK

// folder: Unit6(scaleAndTransferRaw)

FUNCTION_BLOCK "Phase6"   // FB8, SCL
{ S7_Optimized_Access := 'TRUE' }
VERSION : 0.1
   VAR_INPUT
      ena : Bool;
      mode : Int;
      runConveyor : Bool;
      weight : Real;
      transferDone : Bool;
      weightSP : Real;
      resetState : Bool;
   END_VAR
   VAR_OUTPUT
      enaNextStep : Bool;
      weightDone : Bool;
      openValvePerc : Real;
      controlValve : Real;
   END_VAR
   VAR CONSTANT
      factor : Real := 10.0;
      "time" : Time := T#300ms;
   END_VAR
BEGIN
   IF #ena AND NOT #weightDone AND #mode = 1 THEN
       IF ABS_REAL(#weight - #weightSP) > "Recipe".errorWeightRaw1 * #factor THEN
           #openValvePerc := 100;
       ELSE
           #openValvePerc := ABS_REAL(#weight - #weightSP)/"Recipe".errorWeightRaw1 * #factor;
           IF #openValvePerc < "Recipe".openValvePercMin THEN
               #openValvePerc := "Recipe".openValvePercMin;
           END_IF;
       END_IF;
   ELSIF #ena AND #mode = 2 THEN
       #openValvePerc := 50;
   ELSE
       #openValvePerc := 0;
   END_IF;

   IF ABS_REAL( #weight - #weightSP) <= "Recipe".errorWeightRaw1 THEN
       #weightDone := TRUE;
   END_IF;

   IF #weightDone  AND #transferDone THEN
       #enaNextStep := TRUE;
   END_IF;
   IF #resetState THEN
       #enaNextStep := FALSE;
   END_IF;
END_FUNCTION_BLOCK

FUNCTION_BLOCK "Phase7"   // FB9, SCL
{ S7_Optimized_Access := 'TRUE' }
VERSION : 0.1
   VAR_INPUT
      ena : Bool;
      mode : Int;
      runConveyor : Bool;
      weight : Real;
      transferDone : Bool;
      weightSP : Real;
      donePreviousStep : Bool;
      resetState : Bool;
   END_VAR
   VAR_OUTPUT
      enaNextStep : Bool;
      weightDone : Bool;
      openValvePerc : Real;
      controlValve : Real;
   END_VAR
   VAR CONSTANT
      factor : Real := 10.0;
      "time" : Time := T#300ms;
   END_VAR
BEGIN
   IF #ena AND NOT #weightDone AND #mode = 1 AND #donePreviousStep THEN
       IF ABS_REAL(#weight - #weightSP) > "Recipe".errorWeightRaw2 * #factor THEN
           #openValvePerc := 100;
       ELSE
           #openValvePerc := ABS_REAL(#weight - #weightSP) / "Recipe".errorWeightRaw2 * #factor;
           IF #openValvePerc < "Recipe".openValvePercMin THEN
               #openValvePerc := "Recipe".openValvePercMin;
           END_IF;
       END_IF;
   ELSIF #ena AND #mode = 2 THEN
       #openValvePerc := 50;
   ELSE
       #openValvePerc := 0;
   END_IF;

   IF ABS_REAL(#weight - #weightSP) <= "Recipe".errorWeightRaw1 THEN
       #weightDone := TRUE;
   END_IF;

   IF #weightDone AND #transferDone THEN
       #enaNextStep := TRUE;
   END_IF;
   IF #resetState THEN
       #enaNextStep := FALSE;
   END_IF;
END_FUNCTION_BLOCK

FUNCTION_BLOCK "Phase8"   // FB10, SCL
{ S7_Optimized_Access := 'TRUE' }
VERSION : 0.1
   VAR_INPUT
      ena : Bool;
      mode : Int;
      runConveyor : Bool;
      weight : Real;
      transferDone : Bool;
      weightSP : Real;
      resetState : Bool;
   END_VAR
   VAR_OUTPUT
      weightDone : Bool;
      openValvePerc : Real;
      controlValve : Real;
      donePreviousStep : Bool;
      ready : Bool;
   END_VAR
   VAR CONSTANT
      factor : Real := 10.0;
      "time" : Time := T#300ms;
   END_VAR
BEGIN
   IF #ena AND NOT #weightDone AND #mode = 1 AND #donePreviousStep THEN
       IF ABS_REAL(#weight - #weightSP) > "Recipe".errorWeightRaw3 * #factor THEN
           #openValvePerc := 100;
       ELSE
           #openValvePerc := ABS_REAL(#weight - #weightSP) / "Recipe".errorWeightRaw3 * #factor;
           IF #openValvePerc < "Recipe".openValvePercMin THEN
               #openValvePerc := "Recipe".openValvePercMin;
           END_IF;
       END_IF;
   ELSIF #ena AND #mode = 2 THEN
       #openValvePerc := 50;
   ELSE
       #openValvePerc := 0;
   END_IF;

   IF ABS_REAL(#weight - #weightSP) <= "Recipe".errorWeightRaw1 THEN
       #weightDone := TRUE;
   END_IF;

   IF #weightDone AND #transferDone THEN
       #ready := TRUE;
   END_IF;
   IF #resetState THEN
       #ready := FALSE;
   END_IF;
END_FUNCTION_BLOCK

// folder: Unit7(scaleSpice)

FUNCTION_BLOCK "Phase9"   // FB11, SCL
{ S7_Optimized_Access := 'TRUE' }
VERSION : 0.1
   VAR_INPUT
      ena : Bool;
      mode : Int;
      runConveyor : Bool;
      weight : Real;
      weightSP : Real;
      resetState : Bool;
   END_VAR
   VAR_OUTPUT
      openValvePerc : Real;
      controlValve : Real;
      ready : Bool;
   END_VAR
   VAR CONSTANT
      factor : Real := 10.0;
      "time" : Time := T#300ms;
   END_VAR
BEGIN
   IF #ena AND NOT #ready AND #mode = 1 THEN
       IF ABS_REAL(#weight - #weightSP) > "Recipe".errorWeightSpice * #factor THEN
           #openValvePerc := 100;
       ELSE
           #openValvePerc := ABS_REAL(#weight - #weightSP) / "Recipe".errorWeightSpice * #factor;
           IF #openValvePerc < "Recipe".openValvePercMin THEN
               #openValvePerc := "Recipe".openValvePercMin;
           END_IF;
       END_IF;
   ELSIF #ena AND #mode = 2 THEN
       #openValvePerc := 50;
   ELSE
       #openValvePerc := 0;
   END_IF;

   IF ABS_REAL(#weight - #weightSP) <= "Recipe".errorWeightRaw1 THEN
       #ready := TRUE;
   END_IF;

   IF #resetState THEN
       #ready := FALSE;
   END_IF;
END_FUNCTION_BLOCK

// folder: Unit8(scaleWater)

FUNCTION_BLOCK "Phase10"   // FB12, SCL
{ S7_Optimized_Access := 'TRUE' }
VERSION : 0.1
   VAR_INPUT
      ena : Bool;
      mode : Int;
      runConveyor : Bool;
      weight : Real;
      weightSP : Real;
      resetState : Bool;
   END_VAR
   VAR_OUTPUT
      openValvePerc : Real;
      controlValve : Real;
      ready : Bool;
   END_VAR
   VAR CONSTANT
      factor : Real := 10.0;
      "time" : Time := T#300ms;
   END_VAR
BEGIN
   IF #ena AND NOT #ready AND #mode = 1 THEN
       IF ABS_REAL(#weight - #weightSP) > "Recipe".errorWeightSpice * #factor THEN
           #openValvePerc := 100;
       ELSE
           #openValvePerc := ABS_REAL(#weight - #weightSP) / "Recipe".errorWeightSpice * #factor;
           IF #openValvePerc < "Recipe".openValvePercMin THEN
               #openValvePerc := "Recipe".openValvePercMin;
           END_IF;
       END_IF;
   ELSIF #ena AND #mode = 2 THEN 
       #openValvePerc := 50;
   ELSE
       #openValvePerc := 0;
   END_IF;

   IF ABS_REAL(#weight - #weightSP) <= "Recipe".errorWeightRaw1 THEN
       #ready := TRUE;
   END_IF;

   IF #resetState THEN
       #ready := FALSE;
   END_IF;
END_FUNCTION_BLOCK

// folder: Unit9(grindRaws)

FUNCTION_BLOCK "Phase11"   // FB13, LAD
{ S7_Optimized_Access := 'TRUE' }
VERSION : 0.1
   VAR_INPUT
      ena : Bool;
      resetState : Bool;
      "time" : Time;
   END_VAR
   VAR_OUTPUT
      enaNextPhase : Bool;
   END_VAR
BEGIN

REGION Network 1
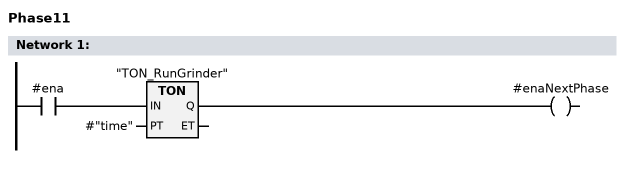
   "TON_RunGrinder".TON(IN := #ena, PT := #"time");
   #enaNextPhase := "TON_RunGrinder".Q;
END_REGION
END_FUNCTION_BLOCK

FUNCTION_BLOCK "Phase12"   // FB14, SCL
{ S7_Optimized_Access := 'TRUE' }
VERSION : 0.1
   VAR_INPUT
      ena : Bool;   // cho phep xa nguyen lieu da nghien
      check : Bool;   // ktra nguyen lieu con tron bon hay ko
      resetState : Bool;
   END_VAR
   VAR_OUTPUT
      ready : Bool;   // tin hieu hoan tat
      openVavle : Bool;   // cho phep mo van xa nguyn lieu
   END_VAR
BEGIN
   IF #ena THEN
       #openVavle := TRUE;
       IF #check THEN
           #ready := TRUE;
       END_IF;
   END_IF;
   IF #resetState THEN
       #ready := FALSE;
   END_IF;
END_FUNCTION_BLOCK

// ===== PLC "PLC_2"  CPU 1211C DC/DC/DC =====

VAR_GLOBAL   // PLC tag table "ControlStep1"
   "highLevelSilo1" AT %Q0.0 : Bool;
   "lowLevelSilo1" AT %Q0.1 : Bool;
   "highLevelSilo2" AT %Q0.2 : Bool;
   "lowLevelSilo2" AT %Q0.3 : Bool;
   "highLevelSilo3" AT %Q0.4 : Bool;
   "lowLevelSilo3" AT %Q0.5 : Bool;
   "highLevelSilo4" AT %Q0.6 : Bool;
   "lowLevelSilo4" AT %Q0.7 : Bool;
   "highLevelSilo5" AT %Q1.0 : Bool;
   "lowLevelSilo5" AT %Q1.1 : Bool;
   "startPumpSilo1" AT %Q1.2 : Bool;
   "stopPumpSilo1" AT %Q1.3 : Bool;
   "startPumpSilo2" AT %Q1.4 : Bool;
   "stopPumpSilo2" AT %Q1.5 : Bool;
   "startPumpSilo3" AT %Q1.6 : Bool;
   "stopPumpSilo3" AT %Q1.7 : Bool;
   "startPumpSilo4" AT %Q2.0 : Bool;
   "stopPumpSilo4" AT %Q2.1 : Bool;
   "startPumpSilo5" AT %Q2.2 : Bool;
   "stopPumpSilo5" AT %Q2.3 : Bool;
   "errorSilo1" AT %I0.0 : Bool;
   "errorSilo2" AT %I0.1 : Bool;
   "errorSilo3" AT %I0.2 : Bool;
   "errorSilo4" AT %I0.3 : Bool;
   "errorSilo5" AT %I0.4 : Bool;
   "levelSilo1" AT %ID6 : Real;
   "levelSilo2" AT %ID10 : Real;
   "levelSilo3" AT %ID14 : Real;
   "levelSilo4" AT %ID18 : Real;
   "levelSilo5" AT %ID22 : Real;
END_VAR

VAR_GLOBAL   // PLC tag table "ControlStep2"
   "weightRaw" AT %ID26 : Real;
   "weightRaw1SP" AT %ID30 : Real;
   "weightRaw2SP" AT %ID34 : Real;
   "weightRaw3SP" AT %ID38 : Real;
   "weightSpice" AT %ID42 : Real;
   "weightSpiceSP" AT %ID46 : Real;
   "weightWater" AT %ID50 : Real;
   "weightWaterSP" AT %ID54 : Real;
   "openRaw1ValvePerc" AT %ID58 : Real;
   "openRaw2ValvePerc" AT %ID62 : Real;
   "openRaw3ValvePerc" AT %ID66 : Real;
   "openSpiceValvePerc" AT %ID70 : Real;
   "openWaterValvePerc" AT %ID74 : Real;
   "transferRawDone" AT %I1.0 : Bool;
END_VAR

VAR_GLOBAL   // PLC tag table "ControlStep3"
   "check" AT %I3.0 : Bool;   // ktra ben trong con nguyen lieu da nghien ko
   "openValve" AT %Q3.0 : Bool;
END_VAR

VAR_GLOBAL   // PLC tag table "ControlStep4"
   "checkSpice" AT %I4.0 : Bool;
   "checkWater" AT %I4.1 : Bool;
   "openValveSpice" AT %Q4.0 : Bool;
   "openValveWater" AT %Q4.1 : Bool;
END_VAR

VAR_GLOBAL   // PLC tag table "ControlStep5"
   "productCheck" AT %I5.0 : Bool;
   "openValveMixer" AT %Q5.0 : Bool;
END_VAR

DATA_BLOCK "Recipe"   // DB1
{ S7_Optimized_Access := 'TRUE' }
VERSION : 0.1
   VAR
      maxLevelSilo1 : Real;   // max cua silo 1
      minLevelSilo1 : Real;   // min cua silo 1
      maxLevelSilo2 : Real;   // max cua silo 2
      minLevelSilo2 : Real;   // min cua silo 2
      maxLevelSilo3 : Real;   // max cua silo 3
      minLevelSilo3 : Real;   // min cua silo 3
      maxLevelSilo4 : Real;   // max cua silo 4
      minLevelSilo4 : Real;   // min cua silo 4
      maxLevelSilo5 : Real;   // max cua silo 5
      minLevelSilo5 : Real;   // min cua silo 5
      weightOfRaw1 : Real;   // khoi luong nguyen lieu 1 can thiet
      weightOfRaw2 : Real;   // khoi luong nguyen lieu 2 can thiet
      weightOfRaw3 : Real;   // khoi luong nguyen lieu 3 can thiet
      weightOfSpice : Real;   // khoi luong gia vi can thiet
      weightOfWater : Real;   // khoi luong nuoc can thiet
      errorWeightRaw1 : Real := 2.5;   // sai so khi do khoi luong nguyen lieu 1
      errorWeightRaw2 : Real := 2.5;   // sai so khi do khoi luong nguyen lieu 2
      errorWeightRaw3 : Real := 2.5;   // sai so khi do khoi luong nguyen lieu 3
      errorWeightSpice : Real := 5.0;   // sai so khi do khoi luong gia vi
      errorWeightWater : Real := 7.0;   // sai so khi do khoi luong nuoc
      openValvePercMin : Real := 10.0;   // % mo van nho nhat de ko gap loi co khi
   END_VAR
BEGIN
END_DATA_BLOCK

DATA_BLOCK "Data"   // DB4
{ S7_Optimized_Access := 'TRUE' }
VERSION : 0.1
   VAR
      state : Int;
      "step" : Int;
      mode : Int;
      set : Bool;
      targetBatches : Int;
      currentBatches : Int;
      silo1Ready : Bool;
      silo2Ready : Bool;
      silo3Ready : Bool;
      silo4Ready : Bool;
      silo5Ready : Bool;
      spiceReady : Bool;
      waterReady : Bool;
      rawReady : Bool;
      grindDone : Bool;
      mixDone : Bool;
      processDone : Bool;
      resetReadyState : Bool;
      enaPumpSilo1 : Bool;
      enaPumpSilo2 : Bool;
      enaPumpSilo3 : Bool;
      enaPumpSilo4 : Bool;
      enaPumpSilo5 : Bool;
      enaScaleRaw1 : Bool;
      enaScaleRaw2 : Bool;
      enaScaleRaw3 : Bool;
      enaScaleSpice : Bool;
      enaScaleWater : Bool;
      runConveyor : Bool;
      runGrinder : Bool;
      runMixer : Bool;
      enaDischargeSpice : Bool;
      enaDischargeWater : Bool;
      enaDischargeMixer : Bool;
      enaNextStep_Raw1 : Bool;
      enaNextStep_Raw2 : Bool;
      weightDoneRaw1 : Bool;
      weightDoneRaw2 : Bool;
      weightDoneRaw3 : Bool;
      enaNextPhase_Grind : Bool;
   END_VAR
BEGIN
END_DATA_BLOCK

DATA_BLOCK "BtnControl"   // DB5
{ S7_Optimized_Access := 'TRUE' }
VERSION : 0.1
   VAR
      start : Bool;
      stop : Bool;
      auto : Bool;
      manu : Bool;
      reset : Bool;
      pause : Bool;
      resume : Bool;
      restart : Bool;
      hold : Bool;
      emerg : Bool;
      abort : Bool;
      alarm : Bool;
      error : Bool;
      btn_silo1 : Bool;
      btn_silo2 : Bool;
      btn_silo3 : Bool;
      btn_silo4 : Bool;
      btn_silo5 : Bool;
      btn_Conveyor : Bool;
      btn_scaleRaw1 : Bool;
      btn_scaleRaw2 : Bool;
      btn_scaleRaw3 : Bool;
      btn_scaleSpice : Bool;
      btn_scaleWater : Bool;
      btn_runGrinder : Bool;
      btn_runMixer : Bool;
      btn_dischargeSpice : Bool;
      btn_dischargeWater : Bool;
      btn_dischargeMixer : Bool;
      btn_ResetReady : Bool;
   END_VAR
BEGIN
END_DATA_BLOCK

DATA_BLOCK "Control_DB"   // DB7
{ S7_Optimized_Access := 'TRUE' }
VERSION : 0.1
// stored: InstanceOfName Control
"Control"
BEGIN
END_DATA_BLOCK

DATA_BLOCK "Process_DB"   // DB8
{ S7_Optimized_Access := 'TRUE' }
VERSION : 0.1
// stored: InstanceOfName Process
"Process"
BEGIN
END_DATA_BLOCK

// folder: DB

DATA_BLOCK "Phase1_DB"   // DB9
{ S7_Optimized_Access := 'TRUE' }
VERSION : 0.1
// stored: InstanceOfName Phase1
"Phase1"
BEGIN
END_DATA_BLOCK

DATA_BLOCK "Phase2_DB"   // DB10
{ S7_Optimized_Access := 'TRUE' }
VERSION : 0.1
// stored: InstanceOfName Phase2
"Phase2"
BEGIN
END_DATA_BLOCK

DATA_BLOCK "Phase3_DB"   // DB11
{ S7_Optimized_Access := 'TRUE' }
VERSION : 0.1
// stored: InstanceOfName Phase3
"Phase3"
BEGIN
END_DATA_BLOCK

DATA_BLOCK "Phase4_DB"   // DB12
{ S7_Optimized_Access := 'TRUE' }
VERSION : 0.1
// stored: InstanceOfName Phase4
"Phase4"
BEGIN
END_DATA_BLOCK

DATA_BLOCK "Phase5_DB"   // DB13
{ S7_Optimized_Access := 'TRUE' }
VERSION : 0.1
// stored: InstanceOfName Phase5
"Phase5"
BEGIN
END_DATA_BLOCK

DATA_BLOCK "Phase6_DB"   // DB14
{ S7_Optimized_Access := 'TRUE' }
VERSION : 0.1
// stored: InstanceOfName Phase6
"Phase6"
BEGIN
END_DATA_BLOCK

DATA_BLOCK "Phase7_DB"   // DB15
{ S7_Optimized_Access := 'TRUE' }
VERSION : 0.1
// stored: InstanceOfName Phase7
"Phase7"
BEGIN
END_DATA_BLOCK

DATA_BLOCK "Phase8_DB"   // DB16
{ S7_Optimized_Access := 'TRUE' }
VERSION : 0.1
// stored: InstanceOfName Phase8
"Phase8"
BEGIN
END_DATA_BLOCK

DATA_BLOCK "Phase9_DB"   // DB17
{ S7_Optimized_Access := 'TRUE' }
VERSION : 0.1
// stored: InstanceOfName Phase9
"Phase9"
BEGIN
END_DATA_BLOCK

DATA_BLOCK "Phase10_DB"   // DB18
{ S7_Optimized_Access := 'TRUE' }
VERSION : 0.1
// stored: InstanceOfName Phase10
"Phase10"
BEGIN
END_DATA_BLOCK

DATA_BLOCK "Phase11_DB"   // DB19
{ S7_Optimized_Access := 'TRUE' }
VERSION : 0.1
// stored: InstanceOfName Phase11
"Phase11"
BEGIN
END_DATA_BLOCK

DATA_BLOCK "Phase12_DB"   // DB20
{ S7_Optimized_Access := 'TRUE' }
VERSION : 0.1
// stored: InstanceOfName Phase12
"Phase12"
BEGIN
END_DATA_BLOCK

DATA_BLOCK "Phase13_DB"   // DB21
{ S7_Optimized_Access := 'TRUE' }
VERSION : 0.1
// stored: InstanceOfName Phase13
"Phase13"
BEGIN
END_DATA_BLOCK

DATA_BLOCK "Phase14_DB"   // DB22
{ S7_Optimized_Access := 'TRUE' }
VERSION : 0.1
// stored: InstanceOfName Phase14
"Phase14"
BEGIN
END_DATA_BLOCK

DATA_BLOCK "Phase15_DB"   // DB23
{ S7_Optimized_Access := 'TRUE' }
VERSION : 0.1
// stored: InstanceOfName Phase15
"Phase15"
BEGIN
END_DATA_BLOCK

DATA_BLOCK "Phase16_DB"   // DB24
{ S7_Optimized_Access := 'TRUE' }
VERSION : 0.1
// stored: InstanceOfName Phase16
"Phase16"
BEGIN
END_DATA_BLOCK

// folder: System blocks/Program resources

DATA_BLOCK "TON_RunMixer"   // DB2
{ S7_Optimized_Access := 'TRUE' }
AUTHOR : Simatic
FAMILY : IEC
NAME : IEC_TMR
VERSION : 1.0
// stored: InstanceOfName IEC_TIMER
"IEC_TIMER"
BEGIN
END_DATA_BLOCK

DATA_BLOCK "TON_RunGrinder"   // DB3
{ S7_Optimized_Access := 'TRUE' }
AUTHOR : Simatic
FAMILY : IEC
NAME : IEC_TMR
VERSION : 1.0
// stored: InstanceOfName IEC_TIMER
"IEC_TIMER"
BEGIN
END_DATA_BLOCK

DATA_BLOCK "TP_ResetReadyState"   // DB6
{ S7_Optimized_Access := 'TRUE' }
AUTHOR : Simatic
FAMILY : IEC
NAME : IEC_TMR
VERSION : 1.0
// stored: InstanceOfName IEC_TIMER
"IEC_TIMER"
BEGIN
END_DATA_BLOCK

// folder: (top level)

FUNCTION_BLOCK "Control"   // FB1, SCL
{ S7_Optimized_Access := 'TRUE' }
VERSION : 0.1
   VAR_INPUT
      start : Bool;
      stop : Bool;
      auto : Bool;
      manu : Bool;
      reset : Bool;
      pause : Bool;
      resume : Bool;
      restart : Bool;
      hold : Bool;
      emerg : Bool;
      abort : Bool;
      alarm : Bool;
      error : Bool;
   END_VAR
   VAR_IN_OUT
      mode : Int;
      state : Int;
      "step" : Int;
   END_VAR
BEGIN
   //chon che do hoat dong
   IF #state = 0 THEN
       IF (#auto AND #manu) OR (NOT #auto AND NOT #manu) THEN
           #mode := 0;
       ELSE
           IF #auto THEN
               #mode := 1;
           END_IF;
           IF #manu THEN
               #mode := 2;
           END_IF;
       END_IF;
   END_IF;

   IF #mode <> 0 THEN
       CASE #state OF
           0:
               IF #start THEN
                   #state := 1;
               END_IF;
           1:
               IF #abort THEN
                   #state := 2;
               ELSIF #stop THEN
                   #state := 3;
               ELSIF #pause THEN
                   #state := 4;
               ELSIF #hold THEN
                   #state := 5;
               ELSIF #step = 6 THEN
                   #state := 6;
               END_IF;
           2, 3, 6:
               IF #reset THEN
                   #state := 0;
               END_IF;
           4:
               IF #resume THEN
                   #state := 1;
               END_IF;
           5:
               IF #restart THEN
                   #state := 1;
               END_IF;

       END_CASE;
   END_IF;
END_FUNCTION_BLOCK

FUNCTION_BLOCK "Process"   // FB2, SCL
{ S7_Optimized_Access := 'TRUE' }
VERSION : 0.1
   VAR_INPUT
      state : Int;   // trang thai hoat dong
      mode : Int;   // che do hoat dong, 1: auto, 2: manu
      set : Bool;   // tin hieu set cac thong so cai dat
      targetBatches : Int;   // So luong me can lam
      currentBatches : Int;   // So luong me hien tai
      silo1Ready : Bool;   // silo 1 da san sang cung cap nguyen lieu
      silo2Ready : Bool;   // silo 2 da san sang cung cap nguyen lieu
      silo3Ready : Bool;   // silo 3 da san sang cung cap nguyen lieu
      silo4Ready : Bool;   // silo 4 da san sang cung cap gia vi
      silo5Ready : Bool;   // silo 5 da san sang cung cap nuoc
      spiceReady : Bool;   // da can xong gia vi
      waterReady : Bool;   // da can xong nuoc
      rawReady : Bool;   // da can xong va dua nguyen lieu vao bon nghien
      grindDone : Bool;   // da nghien xong nguyen lieu
      mixDone : Bool;   // da tron xong nguyen lieu
      processDone : Bool;   // xong quy trinh 1 me
      checkProduct : Bool;   // ktra sp con trong bon tron ko
      btn_resetReady : Bool;   // dkhien reset trang thai ready bang tay (mode manu)
      btn_silo1 : Bool;   // dkhien silo bang tay (mode manu)
      btn_silo2 : Bool;   // dkhien silo bang tay (mode manu)
      btn_silo3 : Bool;   // dkhien silo bang tay (mode manu)
      btn_silo4 : Bool;   // dkhien silo bang tay (mode manu)
      btn_silo5 : Bool;   // dkhien silo bang tay (mode manu)
      btn_runConveyor : Bool;   // dkhien can nguyen lieu bang tay (mode manu)
      btn_scaleRaw1 : Bool;   // xa nguyen lieu raw 1 xuong bang tai bang tay (mode manu)
      btn_scaleRaw2 : Bool;   // xa nguyen lieu raw 2 xuong bang tai bang tay (mode manu)
      btn_scaleRaw3 : Bool;   // xa nguyen lieu raw 3 xuong bang tai bang tay (mode manu)
      btn_scaleSpice : Bool;   // dkhien can gia vi bang tay (mode manu)
      btn_scaleWater : Bool;   // dkhien can nuoc bang tay (mode manu)
      btn_runGrinder : Bool;   // dkhien chay may nghien bang tay (mode manu)
      btn_runMixer : Bool;   // dkhien chay may tron bang tay (mode manu)
      btn_DischargeSpice : Bool;   // dkhien van gia vi bang tay (mode manu)
      btn_DischargeWater : Bool;   // dkhien van nuoc bang tay (mode manu)
      btn_DischargeMixer : Bool;   // dkhien van tron bang tay (mode manu)
   END_VAR
   VAR_OUTPUT
      resetReadyState : Bool;   // tiep tuc lam me moi -> reset lai cac bien ready
      enaPumpSilo1 : Bool;   // cho phep bon 1 bat dau hoat dong
      enaPumpSilo2 : Bool;   // cho phep bon 2 bat dau hoat dong
      enaPumpSilo3 : Bool;   // cho phep bon 3 bat dau hoat dong
      enaPumpSilo4 : Bool;   // cho phep bon 4 bat dau hoat dong
      enaPumpSilo5 : Bool;   // cho phep bon 5 bat dau hoat dong
      enaScaleRaw1 : Bool;   // cho phep can nguyen lieu 1
      enaScaleRaw2 : Bool;   // cho phep can nguyen lieu 2
      enaScaleRaw3 : Bool;   // cho phep can nguyen lieu 3
      enaScaleSpice : Bool;   // cho phep can gia vi
      enaScaleWater : Bool;   // cho phep can nuoc
      runConveyor : Bool;   // chay bang tai
      runGrinder : Bool;   // chay may nghien
      runMixer : Bool;   // chay may tron
      enaDischargeSpice : Bool;   // cho phep xa van gia vi vao may tron
      enaDischargeWater : Bool;   // cho phep xa van nuoc vao may tron
      enaDischargeMixer : Bool;   // cho phep xa hon hop da tron -> hoan thanh 1 batch
   END_VAR
   VAR_IN_OUT
      "step" : Int;
   END_VAR
BEGIN
   IF #state = 1 AND #mode = 1 AND #set THEN
       IF #step = 0 AND #currentBatches < #targetBatches THEN
           #step := 1;
       END_IF;

       CASE #step OF
           1: 
               #enaPumpSilo1 := TRUE;
               #enaPumpSilo2 := TRUE;
               #enaPumpSilo3 := TRUE;
               #enaPumpSilo4 := TRUE;
               #enaPumpSilo5 := TRUE;
               IF #silo1Ready AND #silo2Ready AND #silo3Ready AND #silo4Ready AND #silo5Ready THEN
                   #enaPumpSilo1 := FALSE;
                   #enaPumpSilo2 := FALSE;
                   #enaPumpSilo3 := FALSE;
                   #enaPumpSilo4 := FALSE;
                   #enaPumpSilo5 := FALSE;
                   #step := 2;
               END_IF;

           2: 
               #runConveyor := TRUE;
               #enaScaleRaw1 := TRUE;
               #enaScaleRaw2 := TRUE;
               #enaScaleRaw3 := TRUE;
               #enaScaleWater := TRUE;
               #enaScaleSpice := TRUE;
               IF #rawReady AND #spiceReady AND #waterReady THEN
                   #runConveyor := FALSE;
                   #enaScaleRaw1 := FALSE;
                   #enaScaleRaw2 := FALSE;
                   #enaScaleRaw3 := FALSE;
                   #enaScaleWater := FALSE;
                   #enaScaleSpice := FALSE;
                   #step := 3;
               END_IF;

           3:
               #runGrinder := TRUE;
               IF #grindDone THEN
                   #runGrinder := FALSE;
                   #step := 4;
               END_IF;

           4: 
               #runMixer := TRUE;
               #enaDischargeWater := TRUE; //cho phep mo van, mo bao nhieu % tuy thuoc vao phase 14, 15 quyet dinh
               #enaDischargeSpice := TRUE;
               IF #mixDone THEN
                   #runMixer := FALSE;
                   #enaDischargeWater := FALSE;
                   #enaDischargeSpice := FALSE;
                   #step := 5;
               END_IF;

           5: 
               #enaDischargeMixer := TRUE;
               IF NOT #checkProduct THEN
                   #currentBatches := #currentBatches + 1;
                   #enaDischargeMixer := FALSE;
                   #step := 0;
               END_IF;
               // reset cac bien ready ve FALSE trong 1s -> chac chan bien nao cung dc reset
               "TP_ResetReadyState".TP(IN := NOT #checkProduct AND #processDone,
                                       PT := T#1000ms,
                                       Q => #resetReadyState);
       END_CASE;

   ELSIF #state = 1 AND #mode = 2 AND #set THEN
       #step := 0;
       #resetReadyState := #btn_resetReady;
           //Dk silo
           #enaPumpSilo1 := #btn_silo1;
           #enaPumpSilo2 := #btn_silo2;
           #enaPumpSilo3 := #btn_silo3;
           #enaPumpSilo4 := #btn_silo4;
           #enaPumpSilo5 := #btn_silo5;

           //Dk can va bang tai 
           #runConveyor := #btn_runConveyor;
           #enaScaleRaw1 := #btn_scaleRaw1;
           #enaScaleRaw2 := #btn_scaleRaw2;
           #enaScaleRaw3 := #btn_scaleRaw3;
           #enaScaleWater := #btn_scaleWater;
           #enaScaleSpice := #btn_scaleWater;

           //Dk may nghien va may tron
           #runGrinder := #btn_runGrinder;
           #runMixer := #btn_runMixer;

           //Dong/mo van
           #enaDischargeWater := #btn_DischargeWater;
           #enaDischargeSpice := #btn_DischargeSpice;
           #enaDischargeMixer := #btn_DischargeMixer;
   END_IF;
END_FUNCTION_BLOCK

ORGANIZATION_BLOCK "Main"   // OB1, LAD, ProgramCycle
TITLE = "Main Program Sweep (Cycle)"
{ S7_Optimized_Access := 'TRUE' }
VERSION : 0.1
   VAR_TEMP   // added for the SCL form of the ladder/FBD networks
      _w1 : Bool;
      _w2 : Bool;
   END_VAR
BEGIN

REGION Network 1
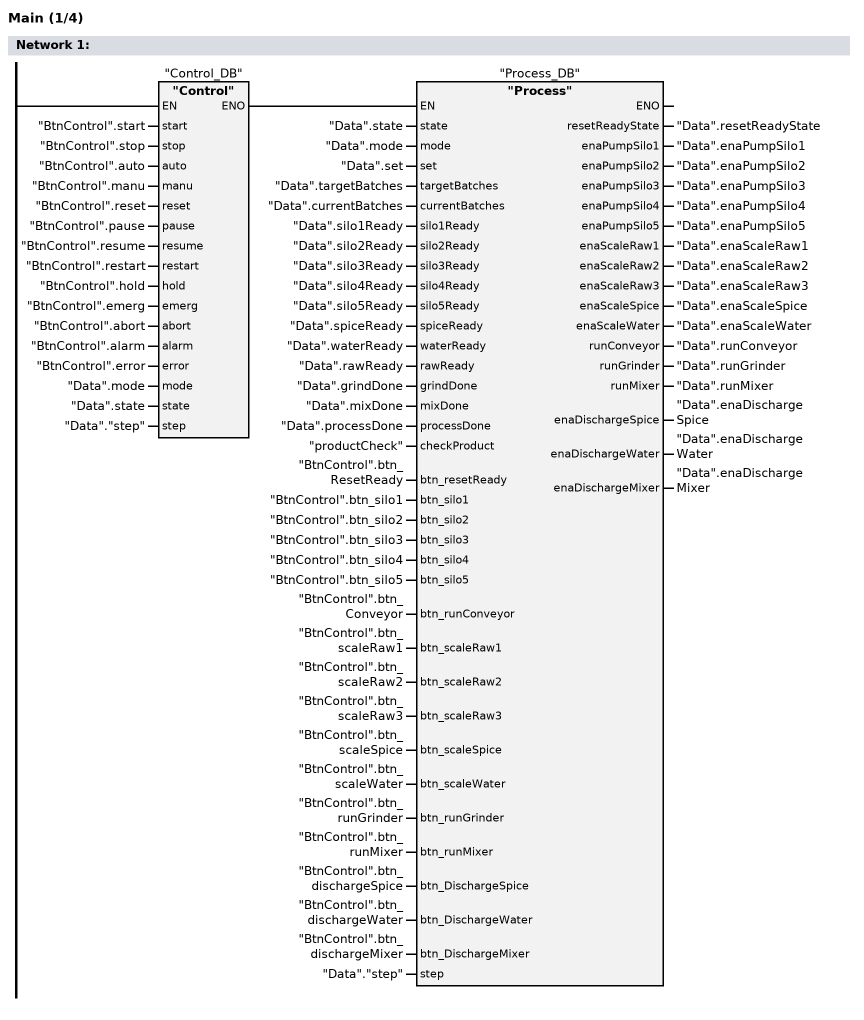
   RUNG wire#powerrail
      "Control_DB"(start := "BtnControl".start, stop := "BtnControl".stop, auto := "BtnControl".auto, manu := "BtnControl".manu, reset := "BtnControl".reset, pause := "BtnControl".pause, resume := "BtnControl".resume, restart := "BtnControl".restart, hold := "BtnControl".hold, emerg := "BtnControl".emerg, abort := "BtnControl".abort, alarm := "BtnControl".alarm, error := "BtnControl".error, mode := "Data".mode, state := "Data".state, "step" := "Data"."step")
      "Process_DB"(state := "Data".state, mode := "Data".mode, set := "Data".set, targetBatches := "Data".targetBatches, currentBatches := "Data".currentBatches, silo1Ready := "Data".silo1Ready, silo2Ready := "Data".silo2Ready, silo3Ready := "Data".silo3Ready, silo4Ready := "Data".silo4Ready, silo5Ready := "Data".silo5Ready, spiceReady := "Data".spiceReady, waterReady := "Data".waterReady, rawReady := "Data".rawReady, grindDone := "Data".grindDone, mixDone := "Data".mixDone, processDone := "Data".processDone, checkProduct := "productCheck", btn_resetReady := "BtnControl".btn_ResetReady, btn_silo1 := "BtnControl".btn_silo1, btn_silo2 := "BtnControl".btn_silo2, btn_silo3 := "BtnControl".btn_silo3, btn_silo4 := "BtnControl".btn_silo4, btn_silo5 := "BtnControl".btn_silo5, btn_runConveyor := "BtnControl".btn_Conveyor, btn_scaleRaw1 := "BtnControl".btn_scaleRaw1, btn_scaleRaw2 := "BtnControl".btn_scaleRaw2, btn_scaleRaw3 := "BtnControl".btn_scaleRaw3, btn_scaleSpice := "BtnControl".btn_scaleSpice, btn_scaleWater := "BtnControl".btn_scaleWater, btn_runGrinder := "BtnControl".btn_runGrinder, btn_runMixer := "BtnControl".btn_runMixer, btn_DischargeSpice := "BtnControl".btn_dischargeSpice, btn_DischargeWater := "BtnControl".btn_dischargeWater, btn_DischargeMixer := "BtnControl".btn_dischargeMixer, "step" := "Data"."step", resetReadyState => "Data".resetReadyState, enaPumpSilo1 => "Data".enaPumpSilo1, enaPumpSilo2 => "Data".enaPumpSilo2, enaPumpSilo3 => "Data".enaPumpSilo3, enaPumpSilo4 => "Data".enaPumpSilo4, enaPumpSilo5 => "Data".enaPumpSilo5, enaScaleRaw1 => "Data".enaScaleRaw1, enaScaleRaw2 => "Data".enaScaleRaw2, enaScaleRaw3 => "Data".enaScaleRaw3, enaScaleSpice => "Data".enaScaleSpice, enaScaleWater => "Data".enaScaleWater, runConveyor => "Data".runConveyor, runGrinder => "Data".runGrinder, runMixer => "Data".runMixer, enaDischargeSpice => "Data".enaDischargeSpice, enaDischargeWater => "Data".enaDischargeWater, enaDischargeMixer => "Data".enaDischargeMixer)
   END_RUNG
   // the same network as SCL:
   "Control_DB"(start := "BtnControl".start,   // "Control"
                stop := "BtnControl".stop,
                auto := "BtnControl".auto,
                manu := "BtnControl".manu,
                reset := "BtnControl".reset,
                pause := "BtnControl".pause,
                resume := "BtnControl".resume,
                restart := "BtnControl".restart,
                hold := "BtnControl".hold,
                emerg := "BtnControl".emerg,
                abort := "BtnControl".abort,
                alarm := "BtnControl".alarm,
                error := "BtnControl".error,
                mode := "Data".mode,
                state := "Data".state,
                "step" := "Data"."step",
                ENO => #_w1);
   IF #_w1 THEN
       "Process_DB"(state := "Data".state,   // "Process"
                    mode := "Data".mode,
                    set := "Data".set,
                    targetBatches := "Data".targetBatches,
                    currentBatches := "Data".currentBatches,
                    silo1Ready := "Data".silo1Ready,
                    silo2Ready := "Data".silo2Ready,
                    silo3Ready := "Data".silo3Ready,
                    silo4Ready := "Data".silo4Ready,
                    silo5Ready := "Data".silo5Ready,
                    spiceReady := "Data".spiceReady,
                    waterReady := "Data".waterReady,
                    rawReady := "Data".rawReady,
                    grindDone := "Data".grindDone,
                    mixDone := "Data".mixDone,
                    processDone := "Data".processDone,
                    checkProduct := "productCheck",
                    btn_resetReady := "BtnControl".btn_ResetReady,
                    btn_silo1 := "BtnControl".btn_silo1,
                    btn_silo2 := "BtnControl".btn_silo2,
                    btn_silo3 := "BtnControl".btn_silo3,
                    btn_silo4 := "BtnControl".btn_silo4,
                    btn_silo5 := "BtnControl".btn_silo5,
                    btn_runConveyor := "BtnControl".btn_Conveyor,
                    btn_scaleRaw1 := "BtnControl".btn_scaleRaw1,
                    btn_scaleRaw2 := "BtnControl".btn_scaleRaw2,
                    btn_scaleRaw3 := "BtnControl".btn_scaleRaw3,
                    btn_scaleSpice := "BtnControl".btn_scaleSpice,
                    btn_scaleWater := "BtnControl".btn_scaleWater,
                    btn_runGrinder := "BtnControl".btn_runGrinder,
                    btn_runMixer := "BtnControl".btn_runMixer,
                    btn_DischargeSpice := "BtnControl".btn_dischargeSpice,
                    btn_DischargeWater := "BtnControl".btn_dischargeWater,
                    btn_DischargeMixer := "BtnControl".btn_dischargeMixer,
                    "step" := "Data"."step",
                    resetReadyState => "Data".resetReadyState,
                    enaPumpSilo1 => "Data".enaPumpSilo1,
                    enaPumpSilo2 => "Data".enaPumpSilo2,
                    enaPumpSilo3 => "Data".enaPumpSilo3,
                    enaPumpSilo4 => "Data".enaPumpSilo4,
                    enaPumpSilo5 => "Data".enaPumpSilo5,
                    enaScaleRaw1 => "Data".enaScaleRaw1,
                    enaScaleRaw2 => "Data".enaScaleRaw2,
                    enaScaleRaw3 => "Data".enaScaleRaw3,
                    enaScaleSpice => "Data".enaScaleSpice,
                    enaScaleWater => "Data".enaScaleWater,
                    runConveyor => "Data".runConveyor,
                    runGrinder => "Data".runGrinder,
                    runMixer => "Data".runMixer,
                    enaDischargeSpice => "Data".enaDischargeSpice,
                    enaDischargeWater => "Data".enaDischargeWater,
                    enaDischargeMixer => "Data".enaDischargeMixer);
   END_IF;
END_REGION

REGION Network 2: Step 1: Fill silos
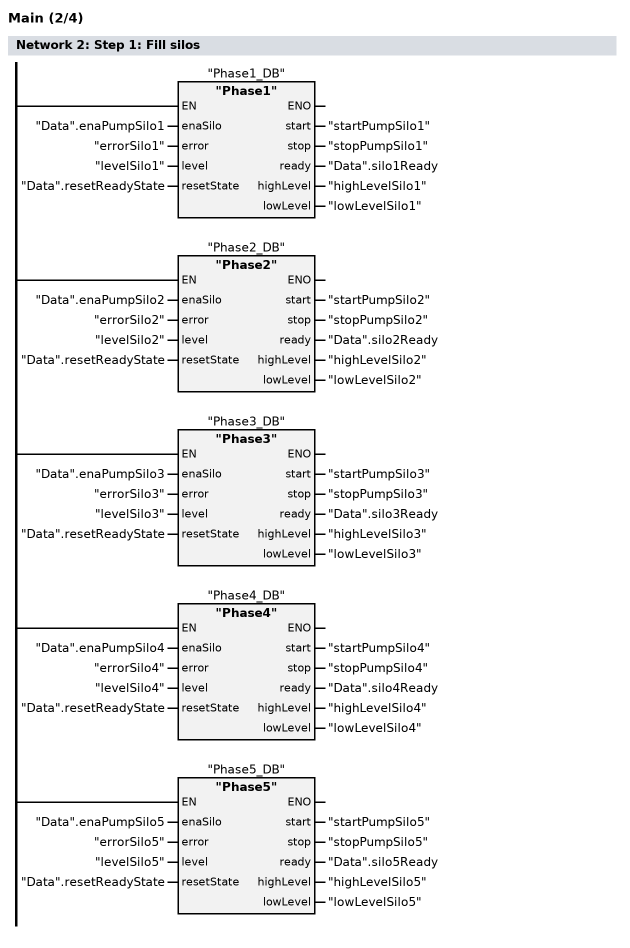
   RUNG wire#powerrail
      "Phase1_DB"(enaSilo := "Data".enaPumpSilo1, error := "errorSilo1", level := "levelSilo1", resetState := "Data".resetReadyState, start => "startPumpSilo1", stop => "stopPumpSilo1", ready => "Data".silo1Ready, highLevel => "highLevelSilo1", lowLevel => "lowLevelSilo1")
   END_RUNG
   RUNG wire#powerrail
      "Phase2_DB"(enaSilo := "Data".enaPumpSilo2, error := "errorSilo2", level := "levelSilo2", resetState := "Data".resetReadyState, start => "startPumpSilo2", stop => "stopPumpSilo2", ready => "Data".silo2Ready, highLevel => "highLevelSilo2", lowLevel => "lowLevelSilo2")
   END_RUNG
   RUNG wire#powerrail
      "Phase3_DB"(enaSilo := "Data".enaPumpSilo3, error := "errorSilo3", level := "levelSilo3", resetState := "Data".resetReadyState, start => "startPumpSilo3", stop => "stopPumpSilo3", ready => "Data".silo3Ready, highLevel => "highLevelSilo3", lowLevel => "lowLevelSilo3")
   END_RUNG
   RUNG wire#powerrail
      "Phase4_DB"(enaSilo := "Data".enaPumpSilo4, error := "errorSilo4", level := "levelSilo4", resetState := "Data".resetReadyState, start => "startPumpSilo4", stop => "stopPumpSilo4", ready => "Data".silo4Ready, highLevel => "highLevelSilo4", lowLevel => "lowLevelSilo4")
   END_RUNG
   RUNG wire#powerrail
      "Phase5_DB"(enaSilo := "Data".enaPumpSilo5, error := "errorSilo5", level := "levelSilo5", resetState := "Data".resetReadyState, start => "startPumpSilo5", stop => "stopPumpSilo5", ready => "Data".silo5Ready, highLevel => "highLevelSilo5", lowLevel => "lowLevelSilo5")
   END_RUNG
   // the same network as SCL:
   "Phase1_DB"(enaSilo := "Data".enaPumpSilo1,   // "Phase1"
               error := "errorSilo1",
               level := "levelSilo1",
               resetState := "Data".resetReadyState,
               start => "startPumpSilo1",
               stop => "stopPumpSilo1",
               ready => "Data".silo1Ready,
               highLevel => "highLevelSilo1",
               lowLevel => "lowLevelSilo1");
   "Phase2_DB"(enaSilo := "Data".enaPumpSilo2,   // "Phase2"
               error := "errorSilo2",
               level := "levelSilo2",
               resetState := "Data".resetReadyState,
               start => "startPumpSilo2",
               stop => "stopPumpSilo2",
               ready => "Data".silo2Ready,
               highLevel => "highLevelSilo2",
               lowLevel => "lowLevelSilo2");
   "Phase3_DB"(enaSilo := "Data".enaPumpSilo3,   // "Phase3"
               error := "errorSilo3",
               level := "levelSilo3",
               resetState := "Data".resetReadyState,
               start => "startPumpSilo3",
               stop => "stopPumpSilo3",
               ready => "Data".silo3Ready,
               highLevel => "highLevelSilo3",
               lowLevel => "lowLevelSilo3");
   "Phase4_DB"(enaSilo := "Data".enaPumpSilo4,   // "Phase4"
               error := "errorSilo4",
               level := "levelSilo4",
               resetState := "Data".resetReadyState,
               start => "startPumpSilo4",
               stop => "stopPumpSilo4",
               ready => "Data".silo4Ready,
               highLevel => "highLevelSilo4",
               lowLevel => "lowLevelSilo4");
   "Phase5_DB"(enaSilo := "Data".enaPumpSilo5,   // "Phase5"
               error := "errorSilo5",
               level := "levelSilo5",
               resetState := "Data".resetReadyState,
               start => "startPumpSilo5",
               stop => "stopPumpSilo5",
               ready => "Data".silo5Ready,
               highLevel => "highLevelSilo5",
               lowLevel => "lowLevelSilo5");
END_REGION

REGION Network 3: Step 2: Transfer and scale
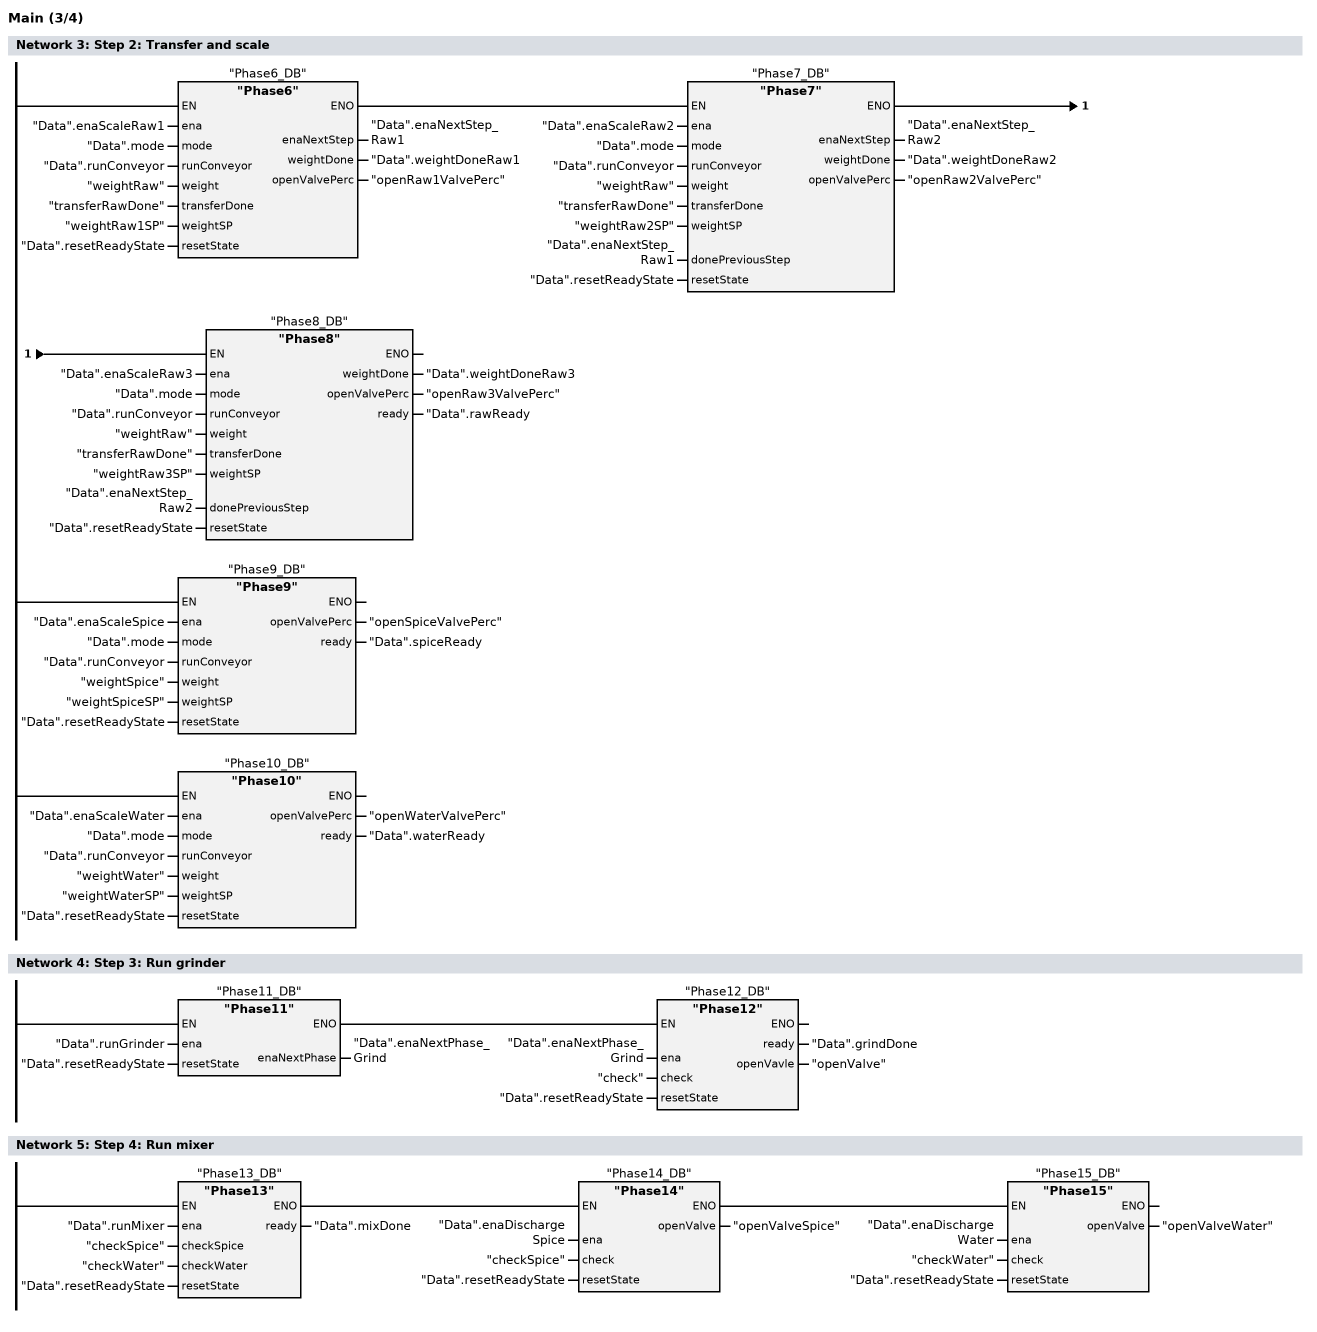
   RUNG wire#powerrail
      "Phase6_DB"(ena := "Data".enaScaleRaw1, mode := "Data".mode, runConveyor := "Data".runConveyor, weight := "weightRaw", transferDone := "transferRawDone", weightSP := "weightRaw1SP", resetState := "Data".resetReadyState, enaNextStep => "Data".enaNextStep_Raw1, weightDone => "Data".weightDoneRaw1, openValvePerc => "openRaw1ValvePerc")
      "Phase7_DB"(ena := "Data".enaScaleRaw2, mode := "Data".mode, runConveyor := "Data".runConveyor, weight := "weightRaw", transferDone := "transferRawDone", weightSP := "weightRaw2SP", donePreviousStep := "Data".enaNextStep_Raw1, resetState := "Data".resetReadyState, enaNextStep => "Data".enaNextStep_Raw2, weightDone => "Data".weightDoneRaw2, openValvePerc => "openRaw2ValvePerc")
      "Phase8_DB"(ena := "Data".enaScaleRaw3, mode := "Data".mode, runConveyor := "Data".runConveyor, weight := "weightRaw", transferDone := "transferRawDone", weightSP := "weightRaw3SP", donePreviousStep := "Data".enaNextStep_Raw2, resetState := "Data".resetReadyState, weightDone => "Data".weightDoneRaw3, openValvePerc => "openRaw3ValvePerc", ready => "Data".rawReady)
   END_RUNG
   RUNG wire#powerrail
      "Phase9_DB"(ena := "Data".enaScaleSpice, mode := "Data".mode, runConveyor := "Data".runConveyor, weight := "weightSpice", weightSP := "weightSpiceSP", resetState := "Data".resetReadyState, openValvePerc => "openSpiceValvePerc", ready => "Data".spiceReady)
   END_RUNG
   RUNG wire#powerrail
      "Phase10_DB"(ena := "Data".enaScaleWater, mode := "Data".mode, runConveyor := "Data".runConveyor, weight := "weightWater", weightSP := "weightWaterSP", resetState := "Data".resetReadyState, openValvePerc => "openWaterValvePerc", ready => "Data".waterReady)
   END_RUNG
   // the same network as SCL:
   "Phase6_DB"(ena := "Data".enaScaleRaw1,   // "Phase6"
               mode := "Data".mode,
               runConveyor := "Data".runConveyor,
               weight := "weightRaw",
               transferDone := "transferRawDone",
               weightSP := "weightRaw1SP",
               resetState := "Data".resetReadyState,
               enaNextStep => "Data".enaNextStep_Raw1,
               weightDone => "Data".weightDoneRaw1,
               openValvePerc => "openRaw1ValvePerc",
               ENO => #_w1);
   "Phase7_DB"(EN := #_w1,   // "Phase7"
               ena := "Data".enaScaleRaw2,
               mode := "Data".mode,
               runConveyor := "Data".runConveyor,
               weight := "weightRaw",
               transferDone := "transferRawDone",
               weightSP := "weightRaw2SP",
               donePreviousStep := "Data".enaNextStep_Raw1,
               resetState := "Data".resetReadyState,
               enaNextStep => "Data".enaNextStep_Raw2,
               weightDone => "Data".weightDoneRaw2,
               openValvePerc => "openRaw2ValvePerc",
               ENO => #_w2);
   IF #_w2 THEN
       "Phase8_DB"(ena := "Data".enaScaleRaw3,   // "Phase8"
                   mode := "Data".mode,
                   runConveyor := "Data".runConveyor,
                   weight := "weightRaw",
                   transferDone := "transferRawDone",
                   weightSP := "weightRaw3SP",
                   donePreviousStep := "Data".enaNextStep_Raw2,
                   resetState := "Data".resetReadyState,
                   weightDone => "Data".weightDoneRaw3,
                   openValvePerc => "openRaw3ValvePerc",
                   ready => "Data".rawReady);
   END_IF;
   "Phase9_DB"(ena := "Data".enaScaleSpice,   // "Phase9"
               mode := "Data".mode,
               runConveyor := "Data".runConveyor,
               weight := "weightSpice",
               weightSP := "weightSpiceSP",
               resetState := "Data".resetReadyState,
               openValvePerc => "openSpiceValvePerc",
               ready => "Data".spiceReady);
   "Phase10_DB"(ena := "Data".enaScaleWater,   // "Phase10"
                mode := "Data".mode,
                runConveyor := "Data".runConveyor,
                weight := "weightWater",
                weightSP := "weightWaterSP",
                resetState := "Data".resetReadyState,
                openValvePerc => "openWaterValvePerc",
                ready => "Data".waterReady);
END_REGION

REGION Network 4: Step 3: Run grinder
   RUNG wire#powerrail
      "Phase11_DB"(ena := "Data".runGrinder, resetState := "Data".resetReadyState, enaNextPhase => "Data".enaNextPhase_Grind)
      "Phase12_DB"(ena := "Data".enaNextPhase_Grind, check := "check", resetState := "Data".resetReadyState, ready => "Data".grindDone, openVavle => "openValve")
   END_RUNG
   // the same network as SCL:
   "Phase11_DB"(ena := "Data".runGrinder,   // "Phase11"
                resetState := "Data".resetReadyState,
                enaNextPhase => "Data".enaNextPhase_Grind,
                ENO => #_w1);
   IF #_w1 THEN
       "Phase12_DB"(ena := "Data".enaNextPhase_Grind,   // "Phase12"
                    check := "check",
                    resetState := "Data".resetReadyState,
                    ready => "Data".grindDone,
                    openVavle => "openValve");
   END_IF;
END_REGION

REGION Network 5: Step 4: Run mixer
   RUNG wire#powerrail
      "Phase13_DB"(ena := "Data".runMixer, checkSpice := "checkSpice", checkWater := "checkWater", resetState := "Data".resetReadyState, ready => "Data".mixDone)
      "Phase14_DB"(ena := "Data".enaDischargeSpice, check := "checkSpice", resetState := "Data".resetReadyState, openValve => "openValveSpice")
      "Phase15_DB"(ena := "Data".enaDischargeWater, check := "checkWater", resetState := "Data".resetReadyState, openValve => "openValveWater")
   END_RUNG
   // the same network as SCL:
   "Phase13_DB"(ena := "Data".runMixer,   // "Phase13"
                checkSpice := "checkSpice",
                checkWater := "checkWater",
                resetState := "Data".resetReadyState,
                ready => "Data".mixDone,
                ENO => #_w1);
   "Phase14_DB"(EN := #_w1,   // "Phase14"
                ena := "Data".enaDischargeSpice,
                check := "checkSpice",
                resetState := "Data".resetReadyState,
                openValve => "openValveSpice",
                ENO => #_w2);
   IF #_w2 THEN
       "Phase15_DB"(ena := "Data".enaDischargeWater,   // "Phase15"
                    check := "checkWater",
                    resetState := "Data".resetReadyState,
                    openValve => "openValveWater");
   END_IF;
END_REGION

REGION Network 6: Step 5: Done
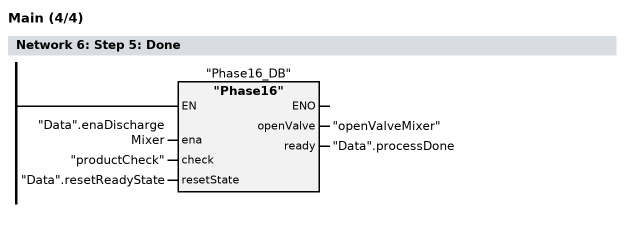
   RUNG wire#powerrail
      "Phase16_DB"(ena := "Data".enaDischargeMixer, check := "productCheck", resetState := "Data".resetReadyState, openValve => "openValveMixer", ready => "Data".processDone)
   END_RUNG
   // the same network as SCL:
   "Phase16_DB"(ena := "Data".enaDischargeMixer,   // "Phase16"
                check := "productCheck",
                resetState := "Data".resetReadyState,
                openValve => "openValveMixer",
                ready => "Data".processDone);
END_REGION
END_ORGANIZATION_BLOCK

// folder: Unit1(prepareSilo1_Raw)

FUNCTION_BLOCK "Phase1"   // FB3, SCL
{ S7_Optimized_Access := 'TRUE' }
VERSION : 0.1
   VAR_INPUT
      enaSilo : Bool;
      error : Bool;
      level : Real;
      resetState : Bool;
   END_VAR
   VAR_OUTPUT
      start : Bool;
      stop : Bool;
      ready : Bool;
      highLevel : Bool;
      lowLevel : Bool;
   END_VAR
BEGIN
   #highLevel := #level >= "Recipe".maxLevelSilo1;
   #lowLevel := #level <= "Recipe".minLevelSilo1;
   #start := #enaSilo AND #lowLevel;
   #stop := #highLevel OR #error;
   #ready := NOT #highLevel AND NOT #lowLevel;
   IF #resetState THEN
       #ready := FALSE;
   END_IF;
END_FUNCTION_BLOCK

// folder: Unit10(mixAndDone)

FUNCTION_BLOCK "Phase13"   // FB15, SCL
{ S7_Optimized_Access := 'TRUE' }
VERSION : 0.1
   VAR_INPUT
      ena : Bool;   // cho phep hoat dong mixer
      checkSpice : Bool;   // ktra da co du gia vi trong bon chua
      checkWater : Bool;   // ktra da co du nuoc trong bon chua
      resetState : Bool;
   END_VAR
   VAR_OUTPUT
      ready : Bool;
   END_VAR
   VAR CONSTANT
      "time" : Time := T#10s;
   END_VAR
BEGIN
   "TON_RunMixer".TON(IN := #ena AND #checkSpice AND #checkWater,
                      PT := #time,
                      Q => #ready);
   IF #resetState THEN
       #ready := FALSE;
   END_IF;
END_FUNCTION_BLOCK

FUNCTION_BLOCK "Phase14"   // FB16, SCL
{ S7_Optimized_Access := 'TRUE' }
VERSION : 0.1
   VAR_INPUT
      ena : Bool;
      check : Bool;   // ktra bon con gia vi ko
      resetState : Bool;
   END_VAR
   VAR_OUTPUT
      openValve : Bool;
   END_VAR
BEGIN
   IF #ena THEN
       #openValve := TRUE;
       IF NOT #check THEN
           #openValve := FALSE;
       END_IF;
   END_IF;
END_FUNCTION_BLOCK

FUNCTION_BLOCK "Phase15"   // FB17, SCL
{ S7_Optimized_Access := 'TRUE' }
VERSION : 0.1
   VAR_INPUT
      ena : Bool;
      check : Bool;   // ktra bon con nuoc ko
      resetState : Bool;
   END_VAR
   VAR_OUTPUT
      openValve : Bool;
   END_VAR
BEGIN
   IF #ena THEN
       #openValve := TRUE;
       IF NOT #check THEN
           #openValve := FALSE;
       END_IF;
   END_IF;
END_FUNCTION_BLOCK

FUNCTION_BLOCK "Phase16"   // FB18, SCL
{ S7_Optimized_Access := 'TRUE' }
VERSION : 0.1
   VAR_INPUT
      ena : Bool;
      check : Bool;   // ktra hon hop con trong bon ko
      resetState : Bool;
   END_VAR
   VAR_OUTPUT
      openValve : Bool;
      ready : Bool;
   END_VAR
BEGIN
   IF #ena THEN
       #openValve := TRUE;
       IF NOT #check THEN
           #openValve := FALSE;
           #ready := TRUE;
       END_IF;
   END_IF;

   IF #resetState THEN
       #ready := FALSE;
   END_IF;
END_FUNCTION_BLOCK

// folder: Unit2(prepareSilo2_Raw)

FUNCTION_BLOCK "Phase2"   // FB4, SCL
{ S7_Optimized_Access := 'TRUE' }
VERSION : 0.1
   VAR_INPUT
      enaSilo : Bool;
      error : Bool;
      level : Real;
      resetState : Bool;
   END_VAR
   VAR_OUTPUT
      start : Bool;
      stop : Bool;
      ready : Bool;
      highLevel : Bool;
      lowLevel : Bool;
   END_VAR
BEGIN
   #highLevel := #level >= "Recipe".maxLevelSilo2;
   #lowLevel := #level <= "Recipe".minLevelSilo2;
   #start := #enaSilo AND #lowLevel;
   #stop := #highLevel OR #error;
   #ready := NOT #highLevel AND NOT #lowLevel;
   IF #resetState THEN
       #ready := FALSE;
   END_IF;
END_FUNCTION_BLOCK

// folder: Unit3(prepareSilo3_Raw)

FUNCTION_BLOCK "Phase3"   // FB5, SCL
{ S7_Optimized_Access := 'TRUE' }
VERSION : 0.1
   VAR_INPUT
      enaSilo : Bool;
      error : Bool;
      level : Real;
      resetState : Bool;
   END_VAR
   VAR_OUTPUT
      start : Bool;
      stop : Bool;
      ready : Bool;
      highLevel : Bool;
      lowLevel : Bool;
   END_VAR
BEGIN
   #highLevel := #level >= "Recipe".maxLevelSilo3;
   #lowLevel := #level <= "Recipe".minLevelSilo3;
   #start := #enaSilo AND #lowLevel;
   #stop := #highLevel OR #error;
   #ready := NOT #highLevel AND NOT #lowLevel;
   IF #resetState THEN
       #ready := FALSE;
   END_IF;
END_FUNCTION_BLOCK

// folder: Unit4(prepareSilo4_Spice)

FUNCTION_BLOCK "Phase4"   // FB6, SCL
{ S7_Optimized_Access := 'TRUE' }
VERSION : 0.1
   VAR_INPUT
      enaSilo : Bool;
      error : Bool;
      level : Real;
      resetState : Bool;
   END_VAR
   VAR_OUTPUT
      start : Bool;
      stop : Bool;
      ready : Bool;
      highLevel : Bool;
      lowLevel : Bool;
   END_VAR
BEGIN
   #highLevel := #level >= "Recipe".maxLevelSilo4;
   #lowLevel := #level <= "Recipe".minLevelSilo4;
   #start := #enaSilo AND #lowLevel;
   #stop := #highLevel OR #error;
   #ready := NOT #highLevel AND NOT #lowLevel;
   IF #resetState THEN
       #ready := FALSE;
   END_IF;
END_FUNCTION_BLOCK

// folder: Unit5(prepareSilo5_Water)

FUNCTION_BLOCK "Phase5"   // FB7, SCL
{ S7_Optimized_Access := 'TRUE' }
VERSION : 0.1
   VAR_INPUT
      enaSilo : Bool;
      error : Bool;
      level : Real;
      resetState : Bool;
   END_VAR
   VAR_OUTPUT
      start : Bool;
      stop : Bool;
      ready : Bool;
      highLevel : Bool;
      lowLevel : Bool;
   END_VAR
BEGIN
   #highLevel := #level >= "Recipe".maxLevelSilo5;
   #lowLevel := #level <= "Recipe".minLevelSilo5;
   #start := #enaSilo AND #lowLevel;
   #stop := #highLevel OR #error;
   #ready := NOT #highLevel AND NOT #lowLevel;
   IF #resetState THEN
       #ready := FALSE;
   END_IF;
END_FUNCTION_BLOCK

// folder: Unit6(scaleAndTransferRaw)

FUNCTION_BLOCK "Phase6"   // FB8, SCL
{ S7_Optimized_Access := 'TRUE' }
VERSION : 0.1
   VAR_INPUT
      ena : Bool;
      mode : Int;
      runConveyor : Bool;
      weight : Real;
      transferDone : Bool;
      weightSP : Real;
      resetState : Bool;
   END_VAR
   VAR_OUTPUT
      enaNextStep : Bool;
      weightDone : Bool;
      openValvePerc : Real;
   END_VAR
   VAR CONSTANT
      factor : Real := 10.0;
      "time" : Time := T#300ms;
   END_VAR
BEGIN
   IF #ena AND NOT #weightDone AND #mode = 1 THEN
       IF ABS_REAL(#weight - #weightSP) > "Recipe".errorWeightRaw1 * #factor THEN
           #openValvePerc := 100;
       ELSE
           #openValvePerc := ABS_REAL(#weight - #weightSP)/"Recipe".errorWeightRaw1 * #factor;
           IF #openValvePerc < "Recipe".openValvePercMin THEN
               #openValvePerc := "Recipe".openValvePercMin;
           END_IF;
       END_IF;
   ELSIF #ena AND #mode = 2 THEN
       #openValvePerc := 50;
   ELSE
       #openValvePerc := 0;
   END_IF;

   IF ABS_REAL( #weight - #weightSP) <= "Recipe".errorWeightRaw1 THEN
       #weightDone := TRUE;
   END_IF;

   IF #weightDone  AND #transferDone THEN
       #enaNextStep := TRUE;
   END_IF;
   IF #resetState THEN
       #enaNextStep := FALSE;
   END_IF;
END_FUNCTION_BLOCK

FUNCTION_BLOCK "Phase7"   // FB9, SCL
{ S7_Optimized_Access := 'TRUE' }
VERSION : 0.1
   VAR_INPUT
      ena : Bool;
      mode : Int;
      runConveyor : Bool;
      weight : Real;
      transferDone : Bool;
      weightSP : Real;
      donePreviousStep : Bool;
      resetState : Bool;
   END_VAR
   VAR_OUTPUT
      enaNextStep : Bool;
      weightDone : Bool;
      openValvePerc : Real;
   END_VAR
   VAR CONSTANT
      factor : Real := 10.0;
      "time" : Time := T#300ms;
   END_VAR
BEGIN
   IF #ena AND NOT #weightDone AND #mode = 1 AND #donePreviousStep THEN
       IF ABS_REAL(#weight - #weightSP) > "Recipe".errorWeightRaw2 * #factor THEN
           #openValvePerc := 100;
       ELSE
           #openValvePerc := ABS_REAL(#weight - #weightSP) / "Recipe".errorWeightRaw2 * #factor;
           IF #openValvePerc < "Recipe".openValvePercMin THEN
               #openValvePerc := "Recipe".openValvePercMin;
           END_IF;
       END_IF;
   ELSIF #ena AND #mode = 2 THEN
       #openValvePerc := 50;
   ELSE
       #openValvePerc := 0;
   END_IF;

   IF ABS_REAL(#weight - #weightSP) <= "Recipe".errorWeightRaw1 THEN
       #weightDone := TRUE;
   END_IF;

   IF #weightDone AND #transferDone THEN
       #enaNextStep := TRUE;
   END_IF;
   IF #resetState THEN
       #enaNextStep := FALSE;
   END_IF;
END_FUNCTION_BLOCK

FUNCTION_BLOCK "Phase8"   // FB10, SCL
{ S7_Optimized_Access := 'TRUE' }
VERSION : 0.1
   VAR_INPUT
      ena : Bool;
      mode : Int;
      runConveyor : Bool;
      weight : Real;
      transferDone : Bool;
      weightSP : Real;
      donePreviousStep : Bool;
      resetState : Bool;
   END_VAR
   VAR_OUTPUT
      weightDone : Bool;
      openValvePerc : Real;
      ready : Bool;
   END_VAR
   VAR CONSTANT
      factor : Real := 10.0;
      "time" : Time := T#300ms;
   END_VAR
BEGIN
   IF #ena AND NOT #weightDone AND #mode = 1 AND #donePreviousStep THEN
       IF ABS_REAL(#weight - #weightSP) > "Recipe".errorWeightRaw3 * #factor THEN
           #openValvePerc := 100;
       ELSE
           #openValvePerc := ABS_REAL(#weight - #weightSP) / "Recipe".errorWeightRaw3 * #factor;
           IF #openValvePerc < "Recipe".openValvePercMin THEN
               #openValvePerc := "Recipe".openValvePercMin;
           END_IF;
       END_IF;
   ELSIF #ena AND #mode = 2 THEN
       #openValvePerc := 50;
   ELSE
       #openValvePerc := 0;
   END_IF;

   IF ABS_REAL(#weight - #weightSP) <= "Recipe".errorWeightRaw1 THEN
       #weightDone := TRUE;
   END_IF;

   IF #weightDone AND #transferDone THEN
       #ready := TRUE;
   END_IF;
   IF #resetState THEN
       #ready := FALSE;
   END_IF;
END_FUNCTION_BLOCK

// folder: Unit7(scaleSpice)

FUNCTION_BLOCK "Phase9"   // FB11, SCL
{ S7_Optimized_Access := 'TRUE' }
VERSION : 0.1
   VAR_INPUT
      ena : Bool;
      mode : Int;
      runConveyor : Bool;
      weight : Real;
      weightSP : Real;
      resetState : Bool;
   END_VAR
   VAR_OUTPUT
      openValvePerc : Real;
      ready : Bool;
   END_VAR
   VAR CONSTANT
      factor : Real := 10.0;
      "time" : Time := T#300ms;
   END_VAR
BEGIN
   IF #ena AND NOT #ready AND #mode = 1 THEN
       IF ABS_REAL(#weight - #weightSP) > "Recipe".errorWeightSpice * #factor THEN
           #openValvePerc := 100;
       ELSE
           #openValvePerc := ABS_REAL(#weight - #weightSP) / "Recipe".errorWeightSpice * #factor;
           IF #openValvePerc < "Recipe".openValvePercMin THEN
               #openValvePerc := "Recipe".openValvePercMin;
           END_IF;
       END_IF;
   ELSIF #ena AND #mode = 2 THEN
       #openValvePerc := 50;
   ELSE
       #openValvePerc := 0;
   END_IF;

   IF ABS_REAL(#weight - #weightSP) <= "Recipe".errorWeightRaw1 THEN
       #ready := TRUE;
   END_IF;

   IF #resetState THEN
       #ready := FALSE;
   END_IF;
END_FUNCTION_BLOCK

// folder: Unit8(scaleWater)

FUNCTION_BLOCK "Phase10"   // FB12, SCL
{ S7_Optimized_Access := 'TRUE' }
VERSION : 0.1
   VAR_INPUT
      ena : Bool;
      mode : Int;
      runConveyor : Bool;
      weight : Real;
      weightSP : Real;
      resetState : Bool;
   END_VAR
   VAR_OUTPUT
      openValvePerc : Real;
      ready : Bool;
   END_VAR
   VAR CONSTANT
      factor : Real := 10.0;
      "time" : Time := T#300ms;
   END_VAR
BEGIN
   IF #ena AND NOT #ready AND #mode = 1 THEN
       IF ABS_REAL(#weight - #weightSP) > "Recipe".errorWeightSpice * #factor THEN
           #openValvePerc := 100;
       ELSE
           #openValvePerc := ABS_REAL(#weight - #weightSP) / "Recipe".errorWeightSpice * #factor;
           IF #openValvePerc < "Recipe".openValvePercMin THEN
               #openValvePerc := "Recipe".openValvePercMin;
           END_IF;
       END_IF;
   ELSIF #ena AND #mode = 2 THEN 
       #openValvePerc := 50;
   ELSE
       #openValvePerc := 0;
   END_IF;

   IF ABS_REAL(#weight - #weightSP) <= "Recipe".errorWeightRaw1 THEN
       #ready := TRUE;
   END_IF;

   IF #resetState THEN
       #ready := FALSE;
   END_IF;
END_FUNCTION_BLOCK

// folder: Unit9(grindRaws)

FUNCTION_BLOCK "Phase11"   // FB13, SCL
{ S7_Optimized_Access := 'TRUE' }
VERSION : 0.1
   VAR_INPUT
      ena : Bool;
      resetState : Bool;
   END_VAR
   VAR_OUTPUT
      enaNextPhase : Bool;
   END_VAR
   VAR CONSTANT
      "time" : Time := T#2s;
   END_VAR
BEGIN
   "TON_RunGrinder".TON(IN := #ena,
                        PT := #time,
                        Q => #enaNextPhase);
   IF #resetState THEN
       #enaNextPhase := FALSE;
   END_IF;
END_FUNCTION_BLOCK

FUNCTION_BLOCK "Phase12"   // FB14, SCL
{ S7_Optimized_Access := 'TRUE' }
VERSION : 0.1
   VAR_INPUT
      ena : Bool;   // cho phep xa nguyen lieu da nghien
      check : Bool;   // ktra nguyen lieu con tron bon hay ko
      resetState : Bool;
   END_VAR
   VAR_OUTPUT
      ready : Bool;   // tin hieu hoan tat
      openVavle : Bool;   // cho phep mo van xa nguyn lieu
   END_VAR
BEGIN
   IF #ena THEN
       #openVavle := TRUE;
       IF #check THEN
           #ready := TRUE;
       END_IF;
   END_IF;
   IF #resetState THEN
       #ready := FALSE;
   END_IF;
END_FUNCTION_BLOCK